LIN {X 0,Y 319.561,Z 300.675,A -85,B 0,C 180,E1 -15416.089,E2 -15416.089} C_VEL
LIN {X 0,Y 319.531,Z 300.681,A -85,B 0,C 180,E1 -15418.933,E2 -15418.933} C_VEL
LIN {X 0,Y 319.51,Z 300.685,A -85,B 0,C 180,E1 -15421.858,E2 -15421.858} C_VEL
LIN {X 0,Y 319.563,Z 300.679,A -85,B 0,C 180,E1 -15425.537,E2 -15425.537} C_VEL
LIN {X 0,Y 319.54,Z 300.681,A -85,B 0,C 180,E1 -15429.663,E2 -15429.663} C_VEL
LIN {X 0,Y 319.497,Z 300.683,A -85,B 0,C 180,E1 -15433.455,E2 -15433.455} C_VEL
LIN {X 0,Y 319.513,Z 300.681,A -85,B 0,C 180,E1 -15437.183,E2 -15437.183} C_VEL
LIN {X 0,Y 319.517,Z 300.684,A -85,B 0,C 180,E1 -15440.366,E2 -15440.366} C_VEL
LIN {X 0,Y 319.508,Z 300.682,A -85,B 0,C 180,E1 -15442.667,E2 -15442.667} C_VEL
LIN {X 0,Y 318.824,Z 300.768,A -85,B 0,C 180,E1 -15443.72,E2 -15443.72} C_VEL
LIN {X 0,Y 315.952,Z 301.126,A -85,B 0,C 180,E1 -15445.434,E2 -15445.434} C_VEL
LIN {X 0,Y 313.541,Z 301.429,A -85,B 0,C 180,E1 -15446.823,E2 -15446.823} C_VEL
LIN {X 0,Y 312.529,Z 301.551,A -85,B 0,C 180,E1 -15447.899,E2 -15447.899} C_VEL
LIN {X 0,Y 312.458,Z 301.56,A -85,B 0,C 180,E1 -15448.263,E2 -15448.263} C_VEL
LIN {X 0,Y 312.537,Z 301.551,A -85,B 0,C 180,E1 -15451.82,E2 -15451.82} C_VEL
LIN {X 0,Y 312.546,Z 301.549,A -85,B 0,C 180,E1 -15454.707,E2 -15454.707} C_VEL
LIN {X 0,Y 312.477,Z 301.558,A -85,B 0,C 180,E1 -15458.908,E2 -15458.908} C_VEL
LIN {X 0,Y 312.519,Z 301.557,A -85,B 0,C 180,E1 -15461.648,E2 -15461.648} C_VEL
LIN {X 0,Y 312.64,Z 301.539,A -85,B 0,C 180,E1 -15465.683,E2 -15465.683} C_VEL
LIN {X 0,Y 312.653,Z 301.536,A -85,B 0,C 180,E1 -15469.64,E2 -15469.64} C_VEL
LIN {X 0,Y 312.798,Z 301.522,A -85,B 0,C 180,E1 -15472.252,E2 -15472.252} C_VEL
LIN {X 0,Y 312.67,Z 301.537,A -85,B 0,C 180,E1 -15474.841,E2 -15474.841} C_VEL
LIN {X 0,Y 312.911,Z 301.504,A -85,B 0,C 180,E1 -15477.425,E2 -15477.425} C_VEL
LIN {X 0,Y 313.034,Z 301.488,A -85,B 0,C 180,E1 -15479.999,E2 -15479.999} C_VEL
LIN {X 0,Y 312.889,Z 301.508,A -85,B 0,C 180,E1 -15482.574,E2 -15482.574} C_VEL
LIN {X 0,Y 312.851,Z 301.511,A -85,B 0,C 180,E1 -15486.448,E2 -15486.448} C_VEL
LIN {X 0,Y 312.712,Z 301.531,A -85,B 0,C 180,E1 -15489.051,E2 -15489.051} C_VEL
LIN {X 0,Y 312.586,Z 301.545,A -85,B 0,C 180,E1 -15492.992,E2 -15492.992} C_VEL
LIN {X 0,Y 312.584,Z 301.549,A -85,B 0,C 180,E1 -15495.652,E2 -15495.652} C_VEL
LIN {X 0,Y 312.565,Z 301.547,A -85,B 0,C 180,E1 -15499.226,E2 -15499.226} C_VEL
LIN {X 0,Y 312.485,Z 301.558,A -85,B 0,C 180,E1 -15502.783,E2 -15502.783} C_VEL
LIN {X 0,Y 312.543,Z 301.551,A -85,B 0,C 180,E1 -15505.931,E2 -15505.931} C_VEL
LIN {X 0,Y 312.467,Z 301.558,A -85,B 0,C 180,E1 -15509.657,E2 -15509.657} C_VEL
LIN {X 0,Y 312.483,Z 301.557,A -85,B 0,C 180,E1 -15513.692,E2 -15513.692} C_VEL
LIN {X 0,Y 312.483,Z 301.56,A -85,B 0,C 180,E1 -15517.39,E2 -15517.39} C_VEL
LIN {X 0,Y 312.457,Z 301.562,A -85,B 0,C 180,E1 -15520.713,E2 -15520.713} C_VEL
LIN {X 0,Y 312.42,Z 301.565,A -85,B 0,C 180,E1 -15524.214,E2 -15524.214} C_VEL
LIN {X 0,Y 312.455,Z 301.564,A -85,B 0,C 180,E1 -15527.924,E2 -15527.924} C_VEL
LIN {X 0,Y 312.452,Z 301.561,A -85,B 0,C 180,E1 -15530.972,E2 -15530.972} C_VEL
LIN {X 0,Y 312.506,Z 301.558,A -85,B 0,C 180,E1 -15534.224,E2 -15534.224} C_VEL
LIN {X 0,Y 312.538,Z 301.702,A -85,B 0,C 180,E1 -15537.345,E2 -15537.345} C_VEL
LIN {X 0,Y 315.451,Z 314.674,A -85,B 0,C 180,E1 -15540.656,E2 -15540.656} C_VEL
LIN {X 0,Y 318.035,Z 327.462,A -85,B 0,C 180,E1 -15543.776,E2 -15543.776} C_VEL
LIN {X 0,Y 316.395,Z 341.128,A -85,B 0,C 180,E1 -15546.784,E2 -15546.784} C_VEL
LIN {X 0,Y 316.002,Z 344.241,A -85,B 0,C 180,E1 -15547.467,E2 -15547.467} C_VEL
LIN {X 0,Y 318.968,Z 375.008,A -85,B 0,C 180,E1 -15548.473,E2 -15548.473} C_VEL
LIN {X 0,Y 317.217,Z 447.196,A -85,B 0,C 180,E1 -15550.426,E2 -15550.426} C_VEL
LIN {X 0,Y 316.799,Z 456.726,A -85,B 0,C 180,E1 -15550.821,E2 -15550.821} C_VEL
LIN {X 0,Y 316.218,Z 466.459,A -85,B 0,C 180,E1 -15551.373,E2 -15551.373} C_VEL
LIN {X 0,Y 315.573,Z 475.191,A -85,B 0,C 180,E1 -15552.005,E2 -15552.005} C_VEL
LIN {X 0,Y 314.745,Z 485.58,A -85,B 0,C 180,E1 -15552.963,E2 -15552.963} C_VEL
LIN {X 0,Y 314.066,Z 494.12,A -85,B 0,C 180,E1 -15553.928,E2 -15553.928} C_VEL
LIN {X 0,Y 313.237,Z 502.921,A -85,B 0,C 180,E1 -15555.13,E2 -15555.13} C_VEL
LIN {X 0,Y 312.614,Z 510.419,A -85,B 0,C 180,E1 -15556.35,E2 -15556.35} C_VEL
LIN {X 0,Y 312.124,Z 517.206,A -85,B 0,C 180,E1 -15557.652,E2 -15557.652} C_VEL
LIN {X 0,Y 311.555,Z 524.228,A -85,B 0,C 180,E1 -15559.278,E2 -15559.278} C_VEL
LIN {X 0,Y 311.202,Z 530.038,A -85,B 0,C 180,E1 -15560.908,E2 -15560.908} C_VEL
LIN {X 0,Y 311.005,Z 535.594,A -85,B 0,C 180,E1 -15562.864,E2 -15562.864} C_VEL
LIN {X 0,Y 310.947,Z 538.236,A -85,B 0,C 180,E1 -15563.973,E2 -15563.973} C_VEL
LIN {X 0,Y 310.901,Z 542.132,A -85,B 0,C 180,E1 -15566.114,E2 -15566.114} C_VEL
LIN {X 0,Y 310.892,Z 543.757,A -85,B 0,C 180,E1 -15567.412,E2 -15567.412} C_VEL
LIN {X 0,Y 311.028,Z 544.971,A -85,B 0,C 180,E1 -15568.708,E2 -15568.708} C_VEL
LIN {X 0,Y 311.069,Z 545.826,A -85,B 0,C 180,E1 -15570.003,E2 -15570.003} C_VEL
LIN {X 0,Y 310.784,Z 545.923,A -85,B 0,C 180,E1 -15572.595,E2 -15572.595} C_VEL
LIN {X 0,Y 310.77,Z 545.451,A -85,B 0,C 180,E1 -15573.892,E2 -15573.892} C_VEL
LIN {X 0,Y 310.772,Z 543.93,A -85,B 0,C 180,E1 -15575.713,E2 -15575.713} C_VEL
LIN {X 0,Y 310.976,Z 541.143,A -85,B 0,C 180,E1 -15577.795,E2 -15577.795} C_VEL
LIN {X 0,Y 311.367,Z 537.429,A -85,B 0,C 180,E1 -15579.748,E2 -15579.748} C_VEL
LIN {X 0,Y 312.047,Z 532.548,A -85,B 0,C 180,E1 -15581.696,E2 -15581.696} C_VEL
LIN {X 0,Y 313.211,Z 526.365,A -85,B 0,C 180,E1 -15583.629,E2 -15583.629} C_VEL
LIN {X 0,Y 314.251,Z 520.119,A -85,B 0,C 180,E1 -15585.236,E2 -15585.236} C_VEL
LIN {X 0,Y 315.608,Z 512.579,A -85,B 0,C 180,E1 -15586.828,E2 -15586.828} C_VEL
LIN {X 0,Y 317.073,Z 504.438,A -85,B 0,C 180,E1 -15588.246,E2 -15588.246} C_VEL
LIN {X 0,Y 318.596,Z 495.771,A -85,B 0,C 180,E1 -15589.491,E2 -15589.491} C_VEL
LIN {X 0,Y 320.051,Z 486.666,A -85,B 0,C 180,E1 -15590.57,E2 -15590.57} C_VEL
LIN {X 0,Y 321.47,Z 477.221,A -85,B 0,C 180,E1 -15591.481,E2 -15591.481} C_VEL
LIN {X 0,Y 322.748,Z 466.457,A -85,B 0,C 180,E1 -15592.316,E2 -15592.316} C_VEL
LIN {X 0,Y 323.729,Z 457.04,A -85,B 0,C 180,E1 -15592.876,E2 -15592.876} C_VEL
LIN {X 0,Y 324.639,Z 446.872,A -85,B 0,C 180,E1 -15593.314,E2 -15593.314} C_VEL
LIN {X 0,Y 325.707,Z 423.932,A -85,B 0,C 180,E1 -15593.992,E2 -15593.992} C_VEL
LIN {X 0,Y 327.83,Z 376.121,A -85,B 0,C 180,E1 -15595.361,E2 -15595.361} C_VEL
LIN {X 0,Y 325.874,Z 360.234,A -85,B 0,C 180,E1 -15596.169,E2 -15596.169} C_VEL
LIN {X 0,Y 322.83,Z 344.326,A -85,B 0,C 180,E1 -15597.151,E2 -15597.151} C_VEL
LIN {X 0,Y 322.58,Z 342.68,A -85,B 0,C 180,E1 -15597.271,E2 -15597.271} C_VEL
LIN {X 0,Y 323.097,Z 338.174,A -85,B 0,C 180,E1 -15598.236,E2 -15598.236} C_VEL
LIN {X 0,Y 321.542,Z 329.706,A -85,B 0,C 180,E1 -15600.485,E2 -15600.485} C_VEL
LIN {X 0,Y 318.939,Z 319.778,A -85,B 0,C 180,E1 -15603.427,E2 -15603.427} C_VEL
LIN {X 0,Y 316.651,Z 312.831,A -85,B 0,C 180,E1 -15605.763,E2 -15605.763} C_VEL
LIN {X 0,Y 313.723,Z 304.747,A -85,B 0,C 180,E1 -15608.846,E2 -15608.846} C_VEL
LIN {X 0,Y 312.479,Z 301.564,A -85,B 0,C 180,E1 -15610.231,E2 -15610.231} C_VEL
LIN {X 0,Y 312.449,Z 301.565,A -85,B 0,C 180,E1 -15613.964,E2 -15613.964} C_VEL
LIN {X 0,Y 312.477,Z 301.559,A -85,B 0,C 180,E1 -15617.918,E2 -15617.918} C_VEL
LIN {X 0,Y 312.53,Z 301.551,A -85,B 0,C 180,E1 -15621.909,E2 -15621.909} C_VEL
LIN {X 0,Y 312.493,Z 301.553,A -85,B 0,C 180,E1 -15625.789,E2 -15625.789} C_VEL
LIN {X 0,Y 312.509,Z 301.548,A -85,B 0,C 180,E1 -15628.853,E2 -15628.853} C_VEL
LIN {X 0,Y 312.559,Z 301.542,A -85,B 0,C 180,E1 -15631.824,E2 -15631.824} C_VEL
LIN {X 0,Y 312.572,Z 301.545,A -85,B 0,C 180,E1 -15634.711,E2 -15634.711} C_VEL
LIN {X 0,Y 312.573,Z 301.551,A -85,B 0,C 180,E1 -15637.529,E2 -15637.529} C_VEL
LIN {X 0,Y 312.621,Z 301.546,A -85,B 0,C 180,E1 -15641.656,E2 -15641.656} C_VEL
LIN {X 0,Y 312.608,Z 301.635,A -85,B 0,C 180,E1 -15644.14,E2 -15644.14} C_VEL
LIN {X 0,Y 315.508,Z 309.164,A -85,B 0,C 180,E1 -15647.13,E2 -15647.13} C_VEL
LIN {X 0,Y 318.415,Z 316.981,A -85,B 0,C 180,E1 -15649.83,E2 -15649.83} C_VEL
LIN {X 0,Y 320.984,Z 325.765,A -85,B 0,C 180,E1 -15652.452,E2 -15652.452} C_VEL
LIN {X 0,Y 322.205,Z 331.817,A -85,B 0,C 180,E1 -15654.054,E2 -15654.054} C_VEL
LIN {X 0,Y 321.513,Z 338.775,A -85,B 0,C 180,E1 -15655.534,E2 -15655.534} C_VEL
LIN {X 0,Y 325.42,Z 357.998,A -85,B 0,C 180,E1 -15656.865,E2 -15656.865} C_VEL
LIN {X 0,Y 327.506,Z 372.724,A -85,B 0,C 180,E1 -15657.73,E2 -15657.73} C_VEL
LIN {X 0,Y 324.419,Z 427.204,A -85,B 0,C 180,E1 -15659.549,E2 -15659.549} C_VEL
LIN {X 0,Y 323.541,Z 438.036,A -85,B 0,C 180,E1 -15660.071,E2 -15660.071} C_VEL
LIN {X 0,Y 322.393,Z 450.107,A -85,B 0,C 180,E1 -15660.906,E2 -15660.906} C_VEL
LIN {X 0,Y 321.132,Z 460.447,A -85,B 0,C 180,E1 -15661.882,E2 -15661.882} C_VEL
LIN {X 0,Y 319.955,Z 468.616,A -85,B 0,C 180,E1 -15662.834,E2 -15662.834} C_VEL
LIN {X 0,Y 318.861,Z 475.526,A -85,B 0,C 180,E1 -15663.792,E2 -15663.792} C_VEL
LIN {X 0,Y 317.505,Z 483.403,A -85,B 0,C 180,E1 -15665.112,E2 -15665.112} C_VEL
LIN {X 0,Y 316.309,Z 489.642,A -85,B 0,C 180,E1 -15666.379,E2 -15666.379} C_VEL
LIN {X 0,Y 315.212,Z 495.003,A -85,B 0,C 180,E1 -15667.689,E2 -15667.689} C_VEL
LIN {X 0,Y 314.311,Z 499.461,A -85,B 0,C 180,E1 -15669.006,E2 -15669.006} C_VEL
LIN {X 0,Y 313.529,Z 503.169,A -85,B 0,C 180,E1 -15670.331,E2 -15670.331} C_VEL
LIN {X 0,Y 312.805,Z 506.225,A -85,B 0,C 180,E1 -15671.667,E2 -15671.667} C_VEL
LIN {X 0,Y 312.252,Z 508.593,A -85,B 0,C 180,E1 -15673.008,E2 -15673.008} C_VEL
LIN {X 0,Y 311.767,Z 510.318,A -85,B 0,C 180,E1 -15674.358,E2 -15674.358} C_VEL
LIN {X 0,Y 311.37,Z 511.487,A -85,B 0,C 180,E1 -15675.716,E2 -15675.716} C_VEL
LIN {X 0,Y 311.102,Z 512.112,A -85,B 0,C 180,E1 -15677.079,E2 -15677.079} C_VEL
LIN {X 0,Y 310.916,Z 512.199,A -85,B 0,C 180,E1 -15678.45,E2 -15678.45} C_VEL
LIN {X 0,Y 310.776,Z 511.681,A -85,B 0,C 180,E1 -15679.83,E2 -15679.83} C_VEL
LIN {X 0,Y 310.787,Z 509.565,A -85,B 0,C 180,E1 -15682.012,E2 -15682.012} C_VEL
LIN {X 0,Y 310.928,Z 507.679,A -85,B 0,C 180,E1 -15683.302,E2 -15683.302} C_VEL
LIN {X 0,Y 311.129,Z 504.922,A -85,B 0,C 180,E1 -15684.702,E2 -15684.702} C_VEL
LIN {X 0,Y 311.489,Z 499.277,A -85,B 0,C 180,E1 -15686.825,E2 -15686.825} C_VEL
LIN {X 0,Y 311.826,Z 494.433,A -85,B 0,C 180,E1 -15688.25,E2 -15688.25} C_VEL
LIN {X 0,Y 312.251,Z 488.495,A -85,B 0,C 180,E1 -15689.681,E2 -15689.681} C_VEL
LIN {X 0,Y 312.852,Z 481.268,A -85,B 0,C 180,E1 -15691.111,E2 -15691.111} C_VEL
LIN {X 0,Y 313.489,Z 473.397,A -85,B 0,C 180,E1 -15692.391,E2 -15692.391} C_VEL
LIN {X 0,Y 314.138,Z 464.159,A -85,B 0,C 180,E1 -15693.623,E2 -15693.623} C_VEL
LIN {X 0,Y 314.847,Z 452.941,A -85,B 0,C 180,E1 -15694.783,E2 -15694.783} C_VEL
LIN {X 0,Y 315.446,Z 444.067,A -85,B 0,C 180,E1 -15695.498,E2 -15695.498} C_VEL
LIN {X 0,Y 315.873,Z 433.915,A -85,B 0,C 180,E1 -15696.13,E2 -15696.13} C_VEL
LIN {X 0,Y 316.224,Z 423.887,A -85,B 0,C 180,E1 -15696.578,E2 -15696.578} C_VEL
LIN {X 0,Y 317.802,Z 367.864,A -85,B 0,C 180,E1 -15698.276,E2 -15698.276} C_VEL
LIN {X 0,Y 314.39,Z 339.94,A -85,B 0,C 180,E1 -15699.315,E2 -15699.315} C_VEL
LIN {X 0,Y 315.823,Z 323.403,A -85,B 0,C 180,E1 -15703.619,E2 -15703.619} C_VEL
LIN {X 0,Y 316.047,Z 319.596,A -85,B 0,C 180,E1 -15704.638,E2 -15704.638} C_VEL
LIN {X 0,Y 313.953,Z 308.571,A -85,B 0,C 180,E1 -15707.814,E2 -15707.814} C_VEL
LIN {X 0,Y 312.499,Z 301.561,A -85,B 0,C 180,E1 -15709.927,E2 -15709.927} C_VEL
LIN {X 0,Y 312.528,Z 301.552,A -85,B 0,C 180,E1 -15714.221,E2 -15714.221} C_VEL
LIN {X 0,Y 312.502,Z 301.556,A -85,B 0,C 180,E1 -15717.334,E2 -15717.334} C_VEL
LIN {X 0,Y 312.486,Z 301.557,A -85,B 0,C 180,E1 -15721.3,E2 -15721.3} C_VEL
LIN {X 0,Y 312.518,Z 301.555,A -85,B 0,C 180,E1 -15724.705,E2 -15724.705} C_VEL
LIN {X 0,Y 312.543,Z 301.549,A -85,B 0,C 180,E1 -15727.525,E2 -15727.525} C_VEL
LIN {X 0,Y 312.571,Z 301.546,A -85,B 0,C 180,E1 -15731.651,E2 -15731.651} C_VEL
LIN {X 0,Y 312.69,Z 301.531,A -85,B 0,C 180,E1 -15735.685,E2 -15735.685} C_VEL
LIN {X 0,Y 312.69,Z 301.533,A -85,B 0,C 180,E1 -15739.64,E2 -15739.64} C_VEL
LIN {X 0,Y 312.801,Z 301.517,A -85,B 0,C 180,E1 -15742.251,E2 -15742.251} C_VEL
LIN {X 0,Y 312.688,Z 301.532,A -85,B 0,C 180,E1 -15744.84,E2 -15744.84} C_VEL
LIN {X 0,Y 312.97,Z 301.496,A -85,B 0,C 180,E1 -15748.711,E2 -15748.711} C_VEL
LIN {X 0,Y 312.969,Z 301.498,A -85,B 0,C 180,E1 -15751.284,E2 -15751.284} C_VEL
LIN {X 0,Y 312.841,Z 301.515,A -85,B 0,C 180,E1 -15756.446,E2 -15756.446} C_VEL
LIN {X 0,Y 312.751,Z 301.524,A -85,B 0,C 180,E1 -15759.047,E2 -15759.047} C_VEL
LIN {X 0,Y 312.633,Z 301.539,A -85,B 0,C 180,E1 -15762.987,E2 -15762.987} C_VEL
LIN {X 0,Y 312.619,Z 301.54,A -85,B 0,C 180,E1 -15765.646,E2 -15765.646} C_VEL
LIN {X 0,Y 312.534,Z 301.551,A -85,B 0,C 180,E1 -15769.708,E2 -15769.708} C_VEL
LIN {X 0,Y 312.515,Z 301.556,A -85,B 0,C 180,E1 -15772.773,E2 -15772.773} C_VEL
LIN {X 0,Y 312.521,Z 301.553,A -85,B 0,C 180,E1 -15775.903,E2 -15775.903} C_VEL
LIN {X 0,Y 312.483,Z 301.56,A -85,B 0,C 180,E1 -15779.65,E2 -15779.65} C_VEL
LIN {X 0,Y 312.505,Z 301.561,A -85,B 0,C 180,E1 -15783.683,E2 -15783.683} C_VEL
LIN {X 0,Y 312.501,Z 301.556,A -85,B 0,C 180,E1 -15787.381,E2 -15787.381} C_VEL
LIN {X 0,Y 312.468,Z 301.559,A -85,B 0,C 180,E1 -15790.704,E2 -15790.704} C_VEL
LIN {X 0,Y 312.427,Z 301.57,A -85,B 0,C 180,E1 -15794.205,E2 -15794.205} C_VEL
LIN {X 0,Y 312.441,Z 301.563,A -85,B 0,C 180,E1 -15797.917,E2 -15797.917} C_VEL
LIN {X 0,Y 312.468,Z 301.562,A -85,B 0,C 180,E1 -15800.966,E2 -15800.966} C_VEL
LIN {X 0,Y 312.498,Z 301.556,A -85,B 0,C 180,E1 -15804.215,E2 -15804.215} C_VEL
LIN {X 0,Y 312.47,Z 301.561,A -85,B 0,C 180,E1 -15807.329,E2 -15807.329} C_VEL
LIN {X 0,Y 312.458,Z 301.56,A -85,B 0,C 180,E1 -15808.263,E2 -15808.263} C_VEL
LIN {X 0,Y 311.806,Z 301.646,A -85,B 0,C 180,E1 -15809.339,E2 -15809.339} C_VEL
LIN {X 0,Y 308.92,Z 302.008,A -85,B 0,C 180,E1 -15811.089,E2 -15811.089} C_VEL
LIN {X 0,Y 306.512,Z 302.307,A -85,B 0,C 180,E1 -15812.509,E2 -15812.509} C_VEL
LIN {X 0,Y 305.551,Z 302.424,A -85,B 0,C 180,E1 -15813.609,E2 -15813.609} C_VEL
LIN {X 0,Y 305.513,Z 302.426,A -85,B 0,C 180,E1 -15813.981,E2 -15813.981} C_VEL
LIN {X 0,Y 305.454,Z 302.433,A -85,B 0,C 180,E1 -15816.974,E2 -15816.974} C_VEL
LIN {X 0,Y 305.472,Z 302.431,A -85,B 0,C 180,E1 -15821.209,E2 -15821.209} C_VEL
LIN {X 0,Y 305.582,Z 302.416,A -85,B 0,C 180,E1 -15825.345,E2 -15825.345} C_VEL
LIN {X 0,Y 305.59,Z 302.416,A -85,B 0,C 180,E1 -15829.397,E2 -15829.397} C_VEL
LIN {X 0,Y 305.741,Z 302.399,A -85,B 0,C 180,E1 -15832.072,E2 -15832.072} C_VEL
LIN {X 0,Y 305.641,Z 302.414,A -85,B 0,C 180,E1 -15834.722,E2 -15834.722} C_VEL
LIN {X 0,Y 305.912,Z 302.38,A -85,B 0,C 180,E1 -15838.683,E2 -15838.683} C_VEL
LIN {X 0,Y 305.909,Z 302.378,A -85,B 0,C 180,E1 -15841.316,E2 -15841.316} C_VEL
LIN {X 0,Y 305.639,Z 302.415,A -85,B 0,C 180,E1 -15845.277,E2 -15845.277} C_VEL
LIN {X 0,Y 305.74,Z 302.398,A -85,B 0,C 180,E1 -15847.927,E2 -15847.927} C_VEL
LIN {X 0,Y 305.555,Z 302.422,A -85,B 0,C 180,E1 -15851.946,E2 -15851.946} C_VEL
LIN {X 0,Y 305.576,Z 302.418,A -85,B 0,C 180,E1 -15855.023,E2 -15855.023} C_VEL
LIN {X 0,Y 305.534,Z 302.422,A -85,B 0,C 180,E1 -15858.785,E2 -15858.785} C_VEL
LIN {X 0,Y 305.446,Z 302.434,A -85,B 0,C 180,E1 -15863.042,E2 -15863.042} C_VEL
LIN {X 0,Y 305.475,Z 302.434,A -85,B 0,C 180,E1 -15866.217,E2 -15866.217} C_VEL
LIN {X 0,Y 305.43,Z 302.436,A -85,B 0,C 180,E1 -15869.043,E2 -15869.043} C_VEL
LIN {X 0,Y 305.398,Z 302.44,A -85,B 0,C 180,E1 -15871.957,E2 -15871.957} C_VEL
LIN {X 0,Y 305.425,Z 302.44,A -85,B 0,C 180,E1 -15875.117,E2 -15875.117} C_VEL
LIN {X 0,Y 305.405,Z 302.44,A -85,B 0,C 180,E1 -15878.53,E2 -15878.53} C_VEL
LIN {X 0,Y 305.396,Z 302.441,A -85,B 0,C 180,E1 -15881.863,E2 -15881.863} C_VEL
LIN {X 0,Y 305.37,Z 302.449,A -85,B 0,C 180,E1 -15885.516,E2 -15885.516} C_VEL
LIN {X 0,Y 305.412,Z 302.44,A -85,B 0,C 180,E1 -15888.147,E2 -15888.147} C_VEL
LIN {X 0,Y 305.43,Z 302.44,A -85,B 0,C 180,E1 -15891.599,E2 -15891.599} C_VEL
LIN {X 0,Y 305.438,Z 302.435,A -85,B 0,C 180,E1 -15894.891,E2 -15894.891} C_VEL
LIN {X 0,Y 305.523,Z 302.623,A -85,B 0,C 180,E1 -15896.99,E2 -15896.99} C_VEL
LIN {X 0,Y 308.337,Z 315.249,A -85,B 0,C 180,E1 -15900.302,E2 -15900.302} C_VEL
LIN {X 0,Y 310.962,Z 328.017,A -85,B 0,C 180,E1 -15903.495,E2 -15903.495} C_VEL
LIN {X 0,Y 310.856,Z 331.099,A -85,B 0,C 180,E1 -15904.207,E2 -15904.207} C_VEL
LIN {X 0,Y 309.07,Z 344.407,A -85,B 0,C 180,E1 -15907.154,E2 -15907.154} C_VEL
LIN {X 0,Y 312.05,Z 375.781,A -85,B 0,C 180,E1 -15908.203,E2 -15908.203} C_VEL
LIN {X 0,Y 310.244,Z 447.06,A -85,B 0,C 180,E1 -15910.183,E2 -15910.183} C_VEL
LIN {X 0,Y 309.818,Z 456.53,A -85,B 0,C 180,E1 -15910.586,E2 -15910.586} C_VEL
LIN {X 0,Y 309.27,Z 465.646,A -85,B 0,C 180,E1 -15911.11,E2 -15911.11} C_VEL
LIN {X 0,Y 308.613,Z 474.48,A -85,B 0,C 180,E1 -15911.757,E2 -15911.757} C_VEL
LIN {X 0,Y 307.777,Z 484.932,A -85,B 0,C 180,E1 -15912.736,E2 -15912.736} C_VEL
LIN {X 0,Y 307.071,Z 493.521,A -85,B 0,C 180,E1 -15913.722,E2 -15913.722} C_VEL
LIN {X 0,Y 306.25,Z 501.887,A -85,B 0,C 180,E1 -15914.876,E2 -15914.876} C_VEL
LIN {X 0,Y 305.678,Z 509.021,A -85,B 0,C 180,E1 -15916.034,E2 -15916.034} C_VEL
LIN {X 0,Y 304.994,Z 517.424,A -85,B 0,C 180,E1 -15917.697,E2 -15917.697} C_VEL
LIN {X 0,Y 304.463,Z 524.347,A -85,B 0,C 180,E1 -15919.362,E2 -15919.362} C_VEL
LIN {X 0,Y 304.155,Z 529.073,A -85,B 0,C 180,E1 -15920.695,E2 -15920.695} C_VEL
LIN {X 0,Y 303.931,Z 534.749,A -85,B 0,C 180,E1 -15922.697,E2 -15922.697} C_VEL
LIN {X 0,Y 303.855,Z 539.118,A -85,B 0,C 180,E1 -15924.695,E2 -15924.695} C_VEL
LIN {X 0,Y 303.839,Z 541.438,A -85,B 0,C 180,E1 -15926.024,E2 -15926.024} C_VEL
LIN {X 0,Y 303.937,Z 544.415,A -85,B 0,C 180,E1 -15928.678,E2 -15928.678} C_VEL
LIN {X 0,Y 303.992,Z 545.32,A -85,B 0,C 180,E1 -15930.003,E2 -15930.003} C_VEL
LIN {X 0,Y 303.702,Z 545.548,A -85,B 0,C 180,E1 -15932.655,E2 -15932.655} C_VEL
LIN {X 0,Y 303.679,Z 545.104,A -85,B 0,C 180,E1 -15933.983,E2 -15933.983} C_VEL
LIN {X 0,Y 303.724,Z 542.731,A -85,B 0,C 180,E1 -15936.646,E2 -15936.646} C_VEL
LIN {X 0,Y 304.028,Z 539.813,A -85,B 0,C 180,E1 -15938.644,E2 -15938.644} C_VEL
LIN {X 0,Y 304.566,Z 535.836,A -85,B 0,C 180,E1 -15940.64,E2 -15940.64} C_VEL
LIN {X 0,Y 305.07,Z 532.626,A -85,B 0,C 180,E1 -15941.968,E2 -15941.968} C_VEL
LIN {X 0,Y 306.304,Z 526.595,A -85,B 0,C 180,E1 -15943.942,E2 -15943.942} C_VEL
LIN {X 0,Y 307.625,Z 519.026,A -85,B 0,C 180,E1 -15945.913,E2 -15945.913} C_VEL
LIN {X 0,Y 308.846,Z 513.058,A -85,B 0,C 180,E1 -15947.208,E2 -15947.208} C_VEL
LIN {X 0,Y 310.591,Z 504.071,A -85,B 0,C 180,E1 -15948.812,E2 -15948.812} C_VEL
LIN {X 0,Y 312.168,Z 495.483,A -85,B 0,C 180,E1 -15950.081,E2 -15950.081} C_VEL
LIN {X 0,Y 313.743,Z 486.47,A -85,B 0,C 180,E1 -15951.175,E2 -15951.175} C_VEL
LIN {X 0,Y 315.206,Z 477.12,A -85,B 0,C 180,E1 -15952.102,E2 -15952.102} C_VEL
LIN {X 0,Y 316.567,Z 466.412,A -85,B 0,C 180,E1 -15952.949,E2 -15952.949} C_VEL
LIN {X 0,Y 317.715,Z 456.324,A -85,B 0,C 180,E1 -15953.55,E2 -15953.55} C_VEL
LIN {X 0,Y 318.616,Z 446.046,A -85,B 0,C 180,E1 -15953.997,E2 -15953.997} C_VEL
LIN {X 0,Y 322.008,Z 377.404,A -85,B 0,C 180,E1 -15956.037,E2 -15956.037} C_VEL
LIN {X 0,Y 320.17,Z 361.869,A -85,B 0,C 180,E1 -15956.854,E2 -15956.854} C_VEL
LIN {X 0,Y 317.028,Z 345.072,A -85,B 0,C 180,E1 -15957.945,E2 -15957.945} C_VEL
LIN {X 0,Y 316.537,Z 342.717,A -85,B 0,C 180,E1 -15958.115,E2 -15958.115} C_VEL
LIN {X 0,Y 316.731,Z 341.02,A -85,B 0,C 180,E1 -15958.493,E2 -15958.493} C_VEL
LIN {X 0,Y 315.465,Z 333.668,A -85,B 0,C 180,E1 -15960.474,E2 -15960.474} C_VEL
LIN {X 0,Y 313.265,Z 324.624,A -85,B 0,C 180,E1 -15963.2,E2 -15963.2} C_VEL
LIN {X 0,Y 311.101,Z 317.62,A -85,B 0,C 180,E1 -15965.585,E2 -15965.585} C_VEL
LIN {X 0,Y 308.345,Z 309.992,A -85,B 0,C 180,E1 -15968.555,E2 -15968.555} C_VEL
LIN {X 0,Y 306.323,Z 305.083,A -85,B 0,C 180,E1 -15970.79,E2 -15970.79} C_VEL
LIN {X 0,Y 305.445,Z 302.44,A -85,B 0,C 180,E1 -15972.128,E2 -15972.128} C_VEL
LIN {X 0,Y 305.416,Z 302.441,A -85,B 0,C 180,E1 -15976.344,E2 -15976.344} C_VEL
LIN {X 0,Y 305.451,Z 302.433,A -85,B 0,C 180,E1 -15979.892,E2 -15979.892} C_VEL
LIN {X 0,Y 305.487,Z 302.43,A -85,B 0,C 180,E1 -15983.627,E2 -15983.627} C_VEL
LIN {X 0,Y 305.452,Z 302.427,A -85,B 0,C 180,E1 -15986.482,E2 -15986.482} C_VEL
LIN {X 0,Y 305.448,Z 302.425,A -85,B 0,C 180,E1 -15989.59,E2 -15989.59} C_VEL
LIN {X 0,Y 305.502,Z 302.424,A -85,B 0,C 180,E1 -15992.608,E2 -15992.608} C_VEL
LIN {X 0,Y 305.496,Z 302.431,A -85,B 0,C 180,E1 -15995.539,E2 -15995.539} C_VEL
LIN {X 0,Y 305.517,Z 302.43,A -85,B 0,C 180,E1 -15999.816,E2 -15999.816} C_VEL
LIN {X 0,Y 305.569,Z 302.583,A -85,B 0,C 180,E1 -16002.344,E2 -16002.344} C_VEL
LIN {X 0,Y 308.406,Z 309.447,A -85,B 0,C 180,E1 -16005.484,E2 -16005.484} C_VEL
LIN {X 0,Y 311.376,Z 317.454,A -85,B 0,C 180,E1 -16008.519,E2 -16008.519} C_VEL
LIN {X 0,Y 313.789,Z 324.958,A -85,B 0,C 180,E1 -16010.981,E2 -16010.981} C_VEL
LIN {X 0,Y 315.403,Z 331.797,A -85,B 0,C 180,E1 -16012.961,E2 -16012.961} C_VEL
LIN {X 0,Y 315.962,Z 335.523,A -85,B 0,C 180,E1 -16013.936,E2 -16013.936} C_VEL
LIN {X 0,Y 315.517,Z 338.867,A -85,B 0,C 180,E1 -16014.649,E2 -16014.649} C_VEL
LIN {X 0,Y 319.253,Z 357.274,A -85,B 0,C 180,E1 -16016.016,E2 -16016.016} C_VEL
LIN {X 0,Y 321.567,Z 372.824,A -85,B 0,C 180,E1 -16016.984,E2 -16016.984} C_VEL
LIN {X 0,Y 318.307,Z 428.295,A -85,B 0,C 180,E1 -16018.924,E2 -16018.924} C_VEL
LIN {X 0,Y 317.36,Z 439.474,A -85,B 0,C 180,E1 -16019.488,E2 -16019.488} C_VEL
LIN {X 0,Y 316.092,Z 451.515,A -85,B 0,C 180,E1 -16020.369,E2 -16020.369} C_VEL
LIN {X 0,Y 314.881,Z 460.932,A -85,B 0,C 180,E1 -16021.28,E2 -16021.28} C_VEL
LIN {X 0,Y 313.636,Z 469.098,A -85,B 0,C 180,E1 -16022.248,E2 -16022.248} C_VEL
LIN {X 0,Y 312.274,Z 477.012,A -85,B 0,C 180,E1 -16023.388,E2 -16023.388} C_VEL
LIN {X 0,Y 310.933,Z 484.094,A -85,B 0,C 180,E1 -16024.621,E2 -16024.621} C_VEL
LIN {X 0,Y 309.723,Z 490.025,A -85,B 0,C 180,E1 -16025.861,E2 -16025.861} C_VEL
LIN {X 0,Y 308.55,Z 495.39,A -85,B 0,C 180,E1 -16027.197,E2 -16027.197} C_VEL
LIN {X 0,Y 307.568,Z 499.866,A -85,B 0,C 180,E1 -16028.542,E2 -16028.542} C_VEL
LIN {X 0,Y 306.334,Z 505.157,A -85,B 0,C 180,E1 -16030.577,E2 -16030.577} C_VEL
LIN {X 0,Y 305.342,Z 509.017,A -85,B 0,C 180,E1 -16032.631,E2 -16032.631} C_VEL
LIN {X 0,Y 304.588,Z 511.445,A -85,B 0,C 180,E1 -16034.704,E2 -16034.704} C_VEL
LIN {X 0,Y 304.217,Z 512.362,A -85,B 0,C 180,E1 -16036.095,E2 -16036.095} C_VEL
LIN {X 0,Y 303.817,Z 512.54,A -85,B 0,C 180,E1 -16038.49,E2 -16038.49} C_VEL
LIN {X 0,Y 303.673,Z 511.58,A -85,B 0,C 180,E1 -16040.314,E2 -16040.314} C_VEL
LIN {X 0,Y 303.711,Z 509.475,A -85,B 0,C 180,E1 -16042.245,E2 -16042.245} C_VEL
LIN {X 0,Y 303.911,Z 506.803,A -85,B 0,C 180,E1 -16043.873,E2 -16043.873} C_VEL
LIN {X 0,Y 304.158,Z 502.737,A -85,B 0,C 180,E1 -16045.696,E2 -16045.696} C_VEL
LIN {X 0,Y 304.522,Z 497.521,A -85,B 0,C 180,E1 -16047.49,E2 -16047.49} C_VEL
LIN {X 0,Y 305.073,Z 490.766,A -85,B 0,C 180,E1 -16049.311,E2 -16049.311} C_VEL
LIN {X 0,Y 305.59,Z 483.904,A -85,B 0,C 180,E1 -16050.779,E2 -16050.779} C_VEL
LIN {X 0,Y 306.277,Z 475.477,A -85,B 0,C 180,E1 -16052.244,E2 -16052.244} C_VEL
LIN {X 0,Y 306.862,Z 467.81,A -85,B 0,C 180,E1 -16053.345,E2 -16053.345} C_VEL
LIN {X 0,Y 307.414,Z 460.172,A -85,B 0,C 180,E1 -16054.262,E2 -16054.262} C_VEL
LIN {X 0,Y 307.989,Z 450.804,A -85,B 0,C 180,E1 -16055.183,E2 -16055.183} C_VEL
LIN {X 0,Y 308.572,Z 441.451,A -85,B 0,C 180,E1 -16055.908,E2 -16055.908} C_VEL
LIN {X 0,Y 309.096,Z 429.632,A -85,B 0,C 180,E1 -16056.595,E2 -16056.595} C_VEL
LIN {X 0,Y 309.611,Z 412.785,A -85,B 0,C 180,E1 -16057.185,E2 -16057.185} C_VEL
LIN {X 0,Y 310.82,Z 367.928,A -85,B 0,C 180,E1 -16058.565,E2 -16058.565} C_VEL
LIN {X 0,Y 307.434,Z 339.917,A -85,B 0,C 180,E1 -16059.644,E2 -16059.644} C_VEL
LIN {X 0,Y 308.924,Z 323.687,A -85,B 0,C 180,E1 -16063.958,E2 -16063.958} C_VEL
LIN {X 0,Y 308.854,Z 319.433,A -85,B 0,C 180,E1 -16065.14,E2 -16065.14} C_VEL
LIN {X 0,Y 306.715,Z 308.538,A -85,B 0,C 180,E1 -16068.358,E2 -16068.358} C_VEL
LIN {X 0,Y 305.467,Z 302.435,A -85,B 0,C 180,E1 -16070.271,E2 -16070.271} C_VEL
LIN {X 0,Y 305.46,Z 302.437,A -85,B 0,C 180,E1 -16073.638,E2 -16073.638} C_VEL
LIN {X 0,Y 305.465,Z 302.432,A -85,B 0,C 180,E1 -16076.484,E2 -16076.484} C_VEL
LIN {X 0,Y 305.418,Z 302.439,A -85,B 0,C 180,E1 -16079.586,E2 -16079.586} C_VEL
LIN {X 0,Y 305.443,Z 302.436,A -85,B 0,C 180,E1 -16082.601,E2 -16082.601} C_VEL
LIN {X 0,Y 305.442,Z 302.434,A -85,B 0,C 180,E1 -16085.533,E2 -16085.533} C_VEL
LIN {X 0,Y 305.485,Z 302.429,A -85,B 0,C 180,E1 -16089.812,E2 -16089.812} C_VEL
LIN {X 0,Y 305.556,Z 302.42,A -85,B 0,C 180,E1 -16093.977,E2 -16093.977} C_VEL
LIN {X 0,Y 305.591,Z 302.418,A -85,B 0,C 180,E1 -16096.703,E2 -16096.703} C_VEL
LIN {X 0,Y 305.758,Z 302.401,A -85,B 0,C 180,E1 -16101.26,E2 -16101.26} C_VEL
LIN {X 0,Y 305.789,Z 302.396,A -85,B 0,C 180,E1 -16103.399,E2 -16103.399} C_VEL
LIN {X 0,Y 305.938,Z 302.372,A -85,B 0,C 180,E1 -16108.681,E2 -16108.681} C_VEL
LIN {X 0,Y 305.937,Z 302.374,A -85,B 0,C 180,E1 -16111.314,E2 -16111.314} C_VEL
LIN {X 0,Y 305.786,Z 302.393,A -85,B 0,C 180,E1 -16116.595,E2 -16116.595} C_VEL
LIN {X 0,Y 305.695,Z 302.402,A -85,B 0,C 180,E1 -16119.257,E2 -16119.257} C_VEL
LIN {X 0,Y 305.585,Z 302.416,A -85,B 0,C 180,E1 -16123.292,E2 -16123.292} C_VEL
LIN {X 0,Y 305.548,Z 302.422,A -85,B 0,C 180,E1 -16126.018,E2 -16126.018} C_VEL
LIN {X 0,Y 305.479,Z 302.43,A -85,B 0,C 180,E1 -16130.183,E2 -16130.183} C_VEL
LIN {X 0,Y 305.466,Z 302.432,A -85,B 0,C 180,E1 -16134.459,E2 -16134.459} C_VEL
LIN {X 0,Y 305.446,Z 302.439,A -85,B 0,C 180,E1 -16137.393,E2 -16137.393} C_VEL
LIN {X 0,Y 305.417,Z 302.436,A -85,B 0,C 180,E1 -16140.408,E2 -16140.408} C_VEL
LIN {X 0,Y 305.449,Z 302.436,A -85,B 0,C 180,E1 -16144.073,E2 -16144.073} C_VEL
LIN {X 0,Y 305.439,Z 302.434,A -85,B 0,C 180,E1 -16146.737,E2 -16146.737} C_VEL
LIN {X 0,Y 305.434,Z 302.436,A -85,B 0,C 180,E1 -16150.594,E2 -16150.594} C_VEL
LIN {X 0,Y 305.402,Z 302.44,A -85,B 0,C 180,E1 -16153.65,E2 -16153.65} C_VEL
LIN {X 0,Y 305.416,Z 302.437,A -85,B 0,C 180,E1 -16157.412,E2 -16157.412} C_VEL
LIN {X 0,Y 305.431,Z 302.436,A -85,B 0,C 180,E1 -16159.887,E2 -16159.887} C_VEL
LIN {X 0,Y 305.432,Z 302.435,A -85,B 0,C 180,E1 -16163.632,E2 -16163.632} C_VEL
LIN {X 0,Y 305.432,Z 302.437,A -85,B 0,C 180,E1 -16166.478,E2 -16166.478} C_VEL
LIN {X 0,Y 305.46,Z 302.435,A -85,B 0,C 180,E1 -16170.947,E2 -16170.947} C_VEL
LIN {X 0,Y 305.513,Z 302.426,A -85,B 0,C 180,E1 -16173.981,E2 -16173.981} C_VEL
LIN {X 0,Y 305.27,Z 302.458,A -85,B 0,C 180,E1 -16174.716,E2 -16174.716} C_VEL
LIN {X 0,Y 303.949,Z 302.625,A -85,B 0,C 180,E1 -16175.802,E2 -16175.802} C_VEL
LIN {X 0,Y 299.522,Z 303.172,A -85,B 0,C 180,E1 -16178.321,E2 -16178.321} C_VEL
LIN {X 0,Y 298.453,Z 303.308,A -85,B 0,C 180,E1 -16179.447,E2 -16179.447} C_VEL
LIN {X 0,Y 298.376,Z 303.314,A -85,B 0,C 180,E1 -16179.829,E2 -16179.829} C_VEL
LIN {X 0,Y 298.437,Z 303.309,A -85,B 0,C 180,E1 -16183.584,E2 -16183.584} C_VEL
LIN {X 0,Y 298.5,Z 303.302,A -85,B 0,C 180,E1 -16186.381,E2 -16186.381} C_VEL
LIN {X 0,Y 298.679,Z 303.277,A -85,B 0,C 180,E1 -16191.161,E2 -16191.161} C_VEL
LIN {X 0,Y 298.738,Z 303.269,A -85,B 0,C 180,E1 -16193.244,E2 -16193.244} C_VEL
LIN {X 0,Y 298.806,Z 303.262,A -85,B 0,C 180,E1 -16197.303,E2 -16197.303} C_VEL
LIN {X 0,Y 298.946,Z 303.243,A -85,B 0,C 180,E1 -16199.999,E2 -16199.999} C_VEL
LIN {X 0,Y 298.789,Z 303.265,A -85,B 0,C 180,E1 -16202.696,E2 -16202.696} C_VEL
LIN {X 0,Y 298.736,Z 303.271,A -85,B 0,C 180,E1 -16206.755,E2 -16206.755} C_VEL
LIN {X 0,Y 298.586,Z 303.293,A -85,B 0,C 180,E1 -16209.483,E2 -16209.483} C_VEL
LIN {X 0,Y 298.502,Z 303.304,A -85,B 0,C 180,E1 -16213.617,E2 -16213.617} C_VEL
LIN {X 0,Y 298.484,Z 303.302,A -85,B 0,C 180,E1 -16216.412,E2 -16216.412} C_VEL
LIN {X 0,Y 298.455,Z 303.307,A -85,B 0,C 180,E1 -16219.648,E2 -16219.648} C_VEL
LIN {X 0,Y 298.387,Z 303.313,A -85,B 0,C 180,E1 -16223.603,E2 -16223.603} C_VEL
LIN {X 0,Y 298.419,Z 303.313,A -85,B 0,C 180,E1 -16226.58,E2 -16226.58} C_VEL
LIN {X 0,Y 298.364,Z 303.315,A -85,B 0,C 180,E1 -16229.646,E2 -16229.646} C_VEL
LIN {X 0,Y 298.355,Z 303.323,A -85,B 0,C 180,E1 -16232.804,E2 -16232.804} C_VEL
LIN {X 0,Y 298.408,Z 303.314,A -85,B 0,C 180,E1 -16236.81,E2 -16236.81} C_VEL
LIN {X 0,Y 298.35,Z 303.322,A -85,B 0,C 180,E1 -16241.09,E2 -16241.09} C_VEL
LIN {X 0,Y 298.37,Z 303.319,A -85,B 0,C 180,E1 -16243.107,E2 -16243.107} C_VEL
LIN {X 0,Y 298.377,Z 303.315,A -85,B 0,C 180,E1 -16246.925,E2 -16246.925} C_VEL
LIN {X 0,Y 298.365,Z 303.316,A -85,B 0,C 180,E1 -16251.014,E2 -16251.014} C_VEL
LIN {X 0,Y 298.381,Z 303.319,A -85,B 0,C 180,E1 -16253.933,E2 -16253.933} C_VEL
LIN {X 0,Y 298.453,Z 303.444,A -85,B 0,C 180,E1 -16256.61,E2 -16256.61} C_VEL
LIN {X 0,Y 301.463,Z 316.996,A -85,B 0,C 180,E1 -16260.24,E2 -16260.24} C_VEL
LIN {X 0,Y 303.853,Z 328.541,A -85,B 0,C 180,E1 -16263.196,E2 -16263.196} C_VEL
LIN {X 0,Y 303.919,Z 331.646,A -85,B 0,C 180,E1 -16263.942,E2 -16263.942} C_VEL
LIN {X 0,Y 302.16,Z 344.254,A -85,B 0,C 180,E1 -16266.822,E2 -16266.822} C_VEL
LIN {X 0,Y 305.138,Z 376.347,A -85,B 0,C 180,E1 -16267.922,E2 -16267.922} C_VEL
LIN {X 0,Y 303.297,Z 446.293,A -85,B 0,C 180,E1 -16269.931,E2 -16269.931} C_VEL
LIN {X 0,Y 302.863,Z 455.875,A -85,B 0,C 180,E1 -16270.343,E2 -16270.343} C_VEL
LIN {X 0,Y 302.257,Z 465.637,A -85,B 0,C 180,E1 -16270.919,E2 -16270.919} C_VEL
LIN {X 0,Y 301.5,Z 475.312,A -85,B 0,C 180,E1 -16271.663,E2 -16271.663} C_VEL
LIN {X 0,Y 300.689,Z 485.557,A -85,B 0,C 180,E1 -16272.667,E2 -16272.667} C_VEL
LIN {X 0,Y 299.981,Z 493.981,A -85,B 0,C 180,E1 -16273.676,E2 -16273.676} C_VEL
LIN {X 0,Y 299.173,Z 501.968,A -85,B 0,C 180,E1 -16274.816,E2 -16274.816} C_VEL
LIN {X 0,Y 298.559,Z 509.24,A -85,B 0,C 180,E1 -16276.042,E2 -16276.042} C_VEL
LIN {X 0,Y 297.864,Z 517.544,A -85,B 0,C 180,E1 -16277.744,E2 -16277.744} C_VEL
LIN {X 0,Y 297.359,Z 524.388,A -85,B 0,C 180,E1 -16279.449,E2 -16279.449} C_VEL
LIN {X 0,Y 297.012,Z 530.025,A -85,B 0,C 180,E1 -16281.156,E2 -16281.156} C_VEL
LIN {X 0,Y 296.871,Z 533.861,A -85,B 0,C 180,E1 -16282.522,E2 -16282.522} C_VEL
LIN {X 0,Y 296.788,Z 538.353,A -85,B 0,C 180,E1 -16284.568,E2 -16284.568} C_VEL
LIN {X 0,Y 296.779,Z 540.685,A -85,B 0,C 180,E1 -16285.929,E2 -16285.929} C_VEL
LIN {X 0,Y 296.846,Z 543.856,A -85,B 0,C 180,E1 -16288.646,E2 -16288.646} C_VEL
LIN {X 0,Y 296.937,Z 544.775,A -85,B 0,C 180,E1 -16290.003,E2 -16290.003} C_VEL
LIN {X 0,Y 296.622,Z 545.172,A -85,B 0,C 180,E1 -16292.719,E2 -16292.719} C_VEL
LIN {X 0,Y 296.592,Z 544.728,A -85,B 0,C 180,E1 -16294.079,E2 -16294.079} C_VEL
LIN {X 0,Y 296.648,Z 542.54,A -85,B 0,C 180,E1 -16296.805,E2 -16296.805} C_VEL
LIN {X 0,Y 296.984,Z 539.734,A -85,B 0,C 180,E1 -16298.85,E2 -16298.85} C_VEL
LIN {X 0,Y 297.571,Z 535.855,A -85,B 0,C 180,E1 -16300.893,E2 -16300.893} C_VEL
LIN {X 0,Y 298.514,Z 530.802,A -85,B 0,C 180,E1 -16302.926,E2 -16302.926} C_VEL
LIN {X 0,Y 299.607,Z 525.62,A -85,B 0,C 180,E1 -16304.607,E2 -16304.607} C_VEL
LIN {X 0,Y 300.975,Z 518.413,A -85,B 0,C 180,E1 -16306.518,E2 -16306.518} C_VEL
LIN {X 0,Y 302.411,Z 511.941,A -85,B 0,C 180,E1 -16307.935,E2 -16307.935} C_VEL
LIN {X 0,Y 304.132,Z 503.871,A -85,B 0,C 180,E1 -16309.402,E2 -16309.402} C_VEL
LIN {X 0,Y 305.791,Z 495.308,A -85,B 0,C 180,E1 -16310.694,E2 -16310.694} C_VEL
LIN {X 0,Y 307.461,Z 486.322,A -85,B 0,C 180,E1 -16311.805,E2 -16311.805} C_VEL
LIN {X 0,Y 309.001,Z 477.013,A -85,B 0,C 180,E1 -16312.747,E2 -16312.747} C_VEL
LIN {X 0,Y 310.428,Z 466.441,A -85,B 0,C 180,E1 -16313.606,E2 -16313.606} C_VEL
LIN {X 0,Y 311.726,Z 455.858,A -85,B 0,C 180,E1 -16314.252,E2 -16314.252} C_VEL
LIN {X 0,Y 312.682,Z 445.697,A -85,B 0,C 180,E1 -16314.704,E2 -16314.704} C_VEL
LIN {X 0,Y 315.413,Z 394.829,A -85,B 0,C 180,E1 -16316.248,E2 -16316.248} C_VEL
LIN {X 0,Y 316.141,Z 377.744,A -85,B 0,C 180,E1 -16316.795,E2 -16316.795} C_VEL
LIN {X 0,Y 314.441,Z 362.812,A -85,B 0,C 180,E1 -16317.619,E2 -16317.619} C_VEL
LIN {X 0,Y 311.231,Z 345.592,A -85,B 0,C 180,E1 -16318.805,E2 -16318.805} C_VEL
LIN {X 0,Y 310.276,Z 342.536,A -85,B 0,C 180,E1 -16319.104,E2 -16319.104} C_VEL
LIN {X 0,Y 308.622,Z 333.962,A -85,B 0,C 180,E1 -16321.584,E2 -16321.584} C_VEL
LIN {X 0,Y 306.451,Z 325.416,A -85,B 0,C 180,E1 -16324.351,E2 -16324.351} C_VEL
LIN {X 0,Y 303.652,Z 316.826,A -85,B 0,C 180,E1 -16327.573,E2 -16327.573} C_VEL
LIN {X 0,Y 301.311,Z 310.626,A -85,B 0,C 180,E1 -16330.322,E2 -16330.322} C_VEL
LIN {X 0,Y 299.694,Z 306.607,A -85,B 0,C 180,E1 -16332.382,E2 -16332.382} C_VEL
LIN {X 0,Y 298.366,Z 303.321,A -85,B 0,C 180,E1 -16334.319,E2 -16334.319} C_VEL
LIN {X 0,Y 298.395,Z 303.317,A -85,B 0,C 180,E1 -16336.92,E2 -16336.92} C_VEL
LIN {X 0,Y 298.414,Z 303.312,A -85,B 0,C 180,E1 -16341.001,E2 -16341.001} C_VEL
LIN {X 0,Y 298.419,Z 303.308,A -85,B 0,C 180,E1 -16343.931,E2 -16343.931} C_VEL
LIN {X 0,Y 298.382,Z 303.308,A -85,B 0,C 180,E1 -16347.984,E2 -16347.984} C_VEL
LIN {X 0,Y 298.447,Z 303.299,A -85,B 0,C 180,E1 -16351.903,E2 -16351.903} C_VEL
LIN {X 0,Y 298.47,Z 303.303,A -85,B 0,C 180,E1 -16354.923,E2 -16354.923} C_VEL
LIN {X 0,Y 298.444,Z 303.309,A -85,B 0,C 180,E1 -16359.316,E2 -16359.316} C_VEL
LIN {X 0,Y 298.516,Z 303.432,A -85,B 0,C 180,E1 -16360.119,E2 -16360.119} C_VEL
LIN {X 0,Y 300.656,Z 308.802,A -85,B 0,C 180,E1 -16363.012,E2 -16363.012} C_VEL
LIN {X 0,Y 302.692,Z 313.449,A -85,B 0,C 180,E1 -16365.203,E2 -16365.203} C_VEL
LIN {X 0,Y 305.924,Z 322.541,A -85,B 0,C 180,E1 -16368.74,E2 -16368.74} C_VEL
LIN {X 0,Y 308.314,Z 330.481,A -85,B 0,C 180,E1 -16371.364,E2 -16371.364} C_VEL
LIN {X 0,Y 309.705,Z 337.936,A -85,B 0,C 180,E1 -16373.486,E2 -16373.486} C_VEL
LIN {X 0,Y 309.607,Z 338.993,A -85,B 0,C 180,E1 -16373.729,E2 -16373.729} C_VEL
LIN {X 0,Y 313.558,Z 358.621,A -85,B 0,C 180,E1 -16375.255,E2 -16375.255} C_VEL
LIN {X 0,Y 315.792,Z 374.119,A -85,B 0,C 180,E1 -16376.274,E2 -16376.274} C_VEL
LIN {X 0,Y 312.364,Z 428.907,A -85,B 0,C 180,E1 -16378.228,E2 -16378.228} C_VEL
LIN {X 0,Y 311.287,Z 440.812,A -85,B 0,C 180,E1 -16378.856,E2 -16378.856} C_VEL
LIN {X 0,Y 309.918,Z 452.405,A -85,B 0,C 180,E1 -16379.748,E2 -16379.748} C_VEL
LIN {X 0,Y 308.658,Z 461.466,A -85,B 0,C 180,E1 -16380.652,E2 -16380.652} C_VEL
LIN {X 0,Y 307.133,Z 470.811,A -85,B 0,C 180,E1 -16381.804,E2 -16381.804} C_VEL
LIN {X 0,Y 305.71,Z 478.531,A -85,B 0,C 180,E1 -16382.966,E2 -16382.966} C_VEL
LIN {X 0,Y 304.003,Z 487.038,A -85,B 0,C 180,E1 -16384.535,E2 -16384.535} C_VEL
LIN {X 0,Y 302.24,Z 494.649,A -85,B 0,C 180,E1 -16386.342,E2 -16386.342} C_VEL
LIN {X 0,Y 300.859,Z 500.312,A -85,B 0,C 180,E1 -16388.058,E2 -16388.058} C_VEL
LIN {X 0,Y 299.65,Z 505.11,A -85,B 0,C 180,E1 -16389.93,E2 -16389.93} C_VEL
LIN {X 0,Y 298.743,Z 508.268,A -85,B 0,C 180,E1 -16391.536,E2 -16391.536} C_VEL
LIN {X 0,Y 298.44,Z 509.449,A -85,B 0,C 180,E1 -16392.237,E2 -16392.237} C_VEL
LIN {X 0,Y 297.578,Z 511.961,A -85,B 0,C 180,E1 -16394.474,E2 -16394.474} C_VEL
LIN {X 0,Y 297.048,Z 512.984,A -85,B 0,C 180,E1 -16396.495,E2 -16396.495} C_VEL
LIN {X 0,Y 296.802,Z 513.089,A -85,B 0,C 180,E1 -16397.929,E2 -16397.929} C_VEL
LIN {X 0,Y 296.644,Z 512.571,A -85,B 0,C 180,E1 -16399.372,E2 -16399.372} C_VEL
LIN {X 0,Y 296.563,Z 511.41,A -85,B 0,C 180,E1 -16400.823,E2 -16400.823} C_VEL
LIN {X 0,Y 296.715,Z 508.577,A -85,B 0,C 180,E1 -16403.045,E2 -16403.045} C_VEL
LIN {X 0,Y 296.996,Z 504.203,A -85,B 0,C 180,E1 -16405.211,E2 -16405.211} C_VEL
LIN {X 0,Y 297.339,Z 499.182,A -85,B 0,C 180,E1 -16407.066,E2 -16407.066} C_VEL
LIN {X 0,Y 297.746,Z 493.602,A -85,B 0,C 180,E1 -16408.701,E2 -16408.701} C_VEL
LIN {X 0,Y 298.205,Z 487.993,A -85,B 0,C 180,E1 -16410.055,E2 -16410.055} C_VEL
LIN {X 0,Y 298.828,Z 480.725,A -85,B 0,C 180,E1 -16411.513,E2 -16411.513} C_VEL
LIN {X 0,Y 299.572,Z 471.286,A -85,B 0,C 180,E1 -16413.056,E2 -16413.056} C_VEL
LIN {X 0,Y 300.346,Z 461.186,A -85,B 0,C 180,E1 -16414.338,E2 -16414.338} C_VEL
LIN {X 0,Y 300.89,Z 452.246,A -85,B 0,C 180,E1 -16415.256,E2 -16415.256} C_VEL
LIN {X 0,Y 301.462,Z 443.714,A -85,B 0,C 180,E1 -16415.959,E2 -16415.959} C_VEL
LIN {X 0,Y 301.948,Z 433.419,A -85,B 0,C 180,E1 -16416.616,E2 -16416.616} C_VEL
LIN {X 0,Y 302.361,Z 421.301,A -85,B 0,C 180,E1 -16417.156,E2 -16417.156} C_VEL
LIN {X 0,Y 303.856,Z 368.389,A -85,B 0,C 180,E1 -16418.845,E2 -16418.845} C_VEL
LIN {X 0,Y 300.479,Z 339.964,A -85,B 0,C 180,E1 -16419.977,E2 -16419.977} C_VEL
LIN {X 0,Y 302.01,Z 324.078,A -85,B 0,C 180,E1 -16424.278,E2 -16424.278} C_VEL
LIN {X 0,Y 301.808,Z 320.4,A -85,B 0,C 180,E1 -16425.329,E2 -16425.329} C_VEL
LIN {X 0,Y 299.651,Z 309.426,A -85,B 0,C 180,E1 -16428.637,E2 -16428.637} C_VEL
LIN {X 0,Y 298.419,Z 303.313,A -85,B 0,C 180,E1 -16430.593,E2 -16430.593} C_VEL
LIN {X 0,Y 298.403,Z 303.314,A -85,B 0,C 180,E1 -16433.929,E2 -16433.929} C_VEL
LIN {X 0,Y 298.393,Z 303.313,A -85,B 0,C 180,E1 -16437.2,E2 -16437.2} C_VEL
LIN {X 0,Y 298.366,Z 303.317,A -85,B 0,C 180,E1 -16440.639,E2 -16440.639} C_VEL
LIN {X 0,Y 298.415,Z 303.31,A -85,B 0,C 180,E1 -16444.917,E2 -16444.917} C_VEL
LIN {X 0,Y 298.396,Z 303.313,A -85,B 0,C 180,E1 -16447.861,E2 -16447.861} C_VEL
LIN {X 0,Y 298.468,Z 303.308,A -85,B 0,C 180,E1 -16450.751,E2 -16450.751} C_VEL
LIN {X 0,Y 298.592,Z 303.291,A -85,B 0,C 180,E1 -16454.993,E2 -16454.993} C_VEL
LIN {X 0,Y 298.588,Z 303.294,A -85,B 0,C 180,E1 -16459.145,E2 -16459.145} C_VEL
LIN {X 0,Y 298.702,Z 303.274,A -85,B 0,C 180,E1 -16461.882,E2 -16461.882} C_VEL
LIN {X 0,Y 298.629,Z 303.282,A -85,B 0,C 180,E1 -16464.596,E2 -16464.596} C_VEL
LIN {X 0,Y 298.906,Z 303.248,A -85,B 0,C 180,E1 -16468.65,E2 -16468.65} C_VEL
LIN {X 0,Y 298.905,Z 303.25,A -85,B 0,C 180,E1 -16471.344,E2 -16471.344} C_VEL
LIN {X 0,Y 298.735,Z 303.27,A -85,B 0,C 180,E1 -16476.752,E2 -16476.752} C_VEL
LIN {X 0,Y 298.626,Z 303.283,A -85,B 0,C 180,E1 -16479.478,E2 -16479.478} C_VEL
LIN {X 0,Y 298.544,Z 303.293,A -85,B 0,C 180,E1 -16483.612,E2 -16483.612} C_VEL
LIN {X 0,Y 298.482,Z 303.304,A -85,B 0,C 180,E1 -16486.408,E2 -16486.408} C_VEL
LIN {X 0,Y 298.441,Z 303.306,A -85,B 0,C 180,E1 -16489.614,E2 -16489.614} C_VEL
LIN {X 0,Y 298.413,Z 303.311,A -85,B 0,C 180,E1 -16493.596,E2 -16493.596} C_VEL
LIN {X 0,Y 298.399,Z 303.312,A -85,B 0,C 180,E1 -16496.577,E2 -16496.577} C_VEL
LIN {X 0,Y 298.381,Z 303.317,A -85,B 0,C 180,E1 -16499.639,E2 -16499.639} C_VEL
LIN {X 0,Y 298.379,Z 303.314,A -85,B 0,C 180,E1 -16502.795,E2 -16502.795} C_VEL
LIN {X 0,Y 298.413,Z 303.31,A -85,B 0,C 180,E1 -16506.798,E2 -16506.798} C_VEL
LIN {X 0,Y 298.365,Z 303.315,A -85,B 0,C 180,E1 -16511.082,E2 -16511.082} C_VEL
LIN {X 0,Y 298.378,Z 303.314,A -85,B 0,C 180,E1 -16513.098,E2 -16513.098} C_VEL
LIN {X 0,Y 298.349,Z 303.319,A -85,B 0,C 180,E1 -16516.91,E2 -16516.91} C_VEL
LIN {X 0,Y 298.369,Z 303.318,A -85,B 0,C 180,E1 -16521.003,E2 -16521.003} C_VEL
LIN {X 0,Y 298.374,Z 303.315,A -85,B 0,C 180,E1 -16523.923,E2 -16523.923} C_VEL
LIN {X 0,Y 298.362,Z 303.32,A -85,B 0,C 180,E1 -16527.195,E2 -16527.195} C_VEL
LIN {X 0,Y 298.397,Z 303.313,A -85,B 0,C 180,E1 -16530.611,E2 -16530.611} C_VEL
LIN {X 0,Y 298.42,Z 303.31,A -85,B 0,C 180,E1 -16533.976,E2 -16533.976} C_VEL
LIN {X 0,Y 298.367,Z 303.319,A -85,B 0,C 180,E1 -16537.859,E2 -16537.859} C_VEL
LIN {X 0,Y 298.376,Z 303.314,A -85,B 0,C 180,E1 -16539.829,E2 -16539.829} C_VEL
LIN {X 0,Y 297.734,Z 303.395,A -85,B 0,C 180,E1 -16540.956,E2 -16540.956} C_VEL
LIN {X 0,Y 294.904,Z 303.747,A -85,B 0,C 180,E1 -16542.791,E2 -16542.791} C_VEL
LIN {X 0,Y 292.513,Z 304.047,A -85,B 0,C 180,E1 -16544.28,E2 -16544.28} C_VEL
LIN {X 0,Y 291.52,Z 304.169,A -85,B 0,C 180,E1 -16545.434,E2 -16545.434} C_VEL
LIN {X 0,Y 291.458,Z 304.178,A -85,B 0,C 180,E1 -16545.824,E2 -16545.824} C_VEL
LIN {X 0,Y 291.53,Z 304.173,A -85,B 0,C 180,E1 -16550.284,E2 -16550.284} C_VEL
LIN {X 0,Y 291.686,Z 304.148,A -85,B 0,C 180,E1 -16553.08,E2 -16553.08} C_VEL
LIN {X 0,Y 291.757,Z 304.14,A -85,B 0,C 180,E1 -16557.238,E2 -16557.238} C_VEL
LIN {X 0,Y 291.904,Z 304.12,A -85,B 0,C 180,E1 -16559.999,E2 -16559.999} C_VEL
LIN {X 0,Y 291.742,Z 304.143,A -85,B 0,C 180,E1 -16562.761,E2 -16562.761} C_VEL
LIN {X 0,Y 291.685,Z 304.15,A -85,B 0,C 180,E1 -16566.919,E2 -16566.919} C_VEL
LIN {X 0,Y 291.528,Z 304.17,A -85,B 0,C 180,E1 -16569.715,E2 -16569.715} C_VEL
LIN {X 0,Y 291.473,Z 304.178,A -85,B 0,C 180,E1 -16573.952,E2 -16573.952} C_VEL
LIN {X 0,Y 291.421,Z 304.183,A -85,B 0,C 180,E1 -16578.27,E2 -16578.27} C_VEL
LIN {X 0,Y 291.322,Z 304.192,A -85,B 0,C 180,E1 -16581.214,E2 -16581.214} C_VEL
LIN {X 0,Y 291.339,Z 304.196,A -85,B 0,C 180,E1 -16584.21,E2 -16584.21} C_VEL
LIN {X 0,Y 291.363,Z 304.188,A -85,B 0,C 180,E1 -16587.277,E2 -16587.277} C_VEL
LIN {X 0,Y 291.285,Z 304.2,A -85,B 0,C 180,E1 -16590.442,E2 -16590.442} C_VEL
LIN {X 0,Y 291.307,Z 304.195,A -85,B 0,C 180,E1 -16593.702,E2 -16593.702} C_VEL
LIN {X 0,Y 291.337,Z 304.195,A -85,B 0,C 180,E1 -16597.256,E2 -16597.256} C_VEL
LIN {X 0,Y 291.297,Z 304.198,A -85,B 0,C 180,E1 -16600.648,E2 -16600.648} C_VEL
LIN {X 0,Y 291.262,Z 304.201,A -85,B 0,C 180,E1 -16604.406,E2 -16604.406} C_VEL
LIN {X 0,Y 291.299,Z 304.197,A -85,B 0,C 180,E1 -16608.409,E2 -16608.409} C_VEL
LIN {X 0,Y 291.314,Z 304.195,A -85,B 0,C 180,E1 -16611.16,E2 -16611.16} C_VEL
LIN {X 0,Y 291.333,Z 304.193,A -85,B 0,C 180,E1 -16614.63,E2 -16614.63} C_VEL
LIN {X 0,Y 291.409,Z 304.279,A -85,B 0,C 180,E1 -16616.217,E2 -16616.217} C_VEL
LIN {X 0,Y 294.383,Z 317.729,A -85,B 0,C 180,E1 -16619.917,E2 -16619.917} C_VEL
LIN {X 0,Y 296.996,Z 330.572,A -85,B 0,C 180,E1 -16623.287,E2 -16623.287} C_VEL
LIN {X 0,Y 296.118,Z 338.172,A -85,B 0,C 180,E1 -16625.091,E2 -16625.091} C_VEL
LIN {X 0,Y 295.231,Z 344.133,A -85,B 0,C 180,E1 -16626.492,E2 -16626.492} C_VEL
LIN {X 0,Y 297.993,Z 373.961,A -85,B 0,C 180,E1 -16627.548,E2 -16627.548} C_VEL
LIN {X 0,Y 298.108,Z 380.004,A -85,B 0,C 180,E1 -16627.739,E2 -16627.739} C_VEL
LIN {X 0,Y 296.305,Z 446.57,A -85,B 0,C 180,E1 -16629.708,E2 -16629.708} C_VEL
LIN {X 0,Y 295.808,Z 456.734,A -85,B 0,C 180,E1 -16630.171,E2 -16630.171} C_VEL
LIN {X 0,Y 295.234,Z 465.612,A -85,B 0,C 180,E1 -16630.718,E2 -16630.718} C_VEL
LIN {X 0,Y 294.552,Z 474.302,A -85,B 0,C 180,E1 -16631.395,E2 -16631.395} C_VEL
LIN {X 0,Y 293.727,Z 484.679,A -85,B 0,C 180,E1 -16632.422,E2 -16632.422} C_VEL
LIN {X 0,Y 292.947,Z 493.704,A -85,B 0,C 180,E1 -16633.526,E2 -16633.526} C_VEL
LIN {X 0,Y 292.052,Z 502.525,A -85,B 0,C 180,E1 -16634.834,E2 -16634.834} C_VEL
LIN {X 0,Y 291.426,Z 509.453,A -85,B 0,C 180,E1 -16636.049,E2 -16636.049} C_VEL
LIN {X 0,Y 290.893,Z 516.221,A -85,B 0,C 180,E1 -16637.445,E2 -16637.445} C_VEL
LIN {X 0,Y 290.317,Z 523.225,A -85,B 0,C 180,E1 -16639.19,E2 -16639.19} C_VEL
LIN {X 0,Y 289.962,Z 529.01,A -85,B 0,C 180,E1 -16640.939,E2 -16640.939} C_VEL
LIN {X 0,Y 289.814,Z 532.92,A -85,B 0,C 180,E1 -16642.339,E2 -16642.339} C_VEL
LIN {X 0,Y 289.703,Z 537.575,A -85,B 0,C 180,E1 -16644.435,E2 -16644.435} C_VEL
LIN {X 0,Y 289.72,Z 539.923,A -85,B 0,C 180,E1 -16645.83,E2 -16645.83} C_VEL
LIN {X 0,Y 289.756,Z 543.294,A -85,B 0,C 180,E1 -16648.613,E2 -16648.613} C_VEL
LIN {X 0,Y 289.882,Z 544.212,A -85,B 0,C 180,E1 -16650.003,E2 -16650.003} C_VEL
LIN {X 0,Y 289.543,Z 544.796,A -85,B 0,C 180,E1 -16652.785,E2 -16652.785} C_VEL
LIN {X 0,Y 289.507,Z 544.353,A -85,B 0,C 180,E1 -16654.179,E2 -16654.179} C_VEL
LIN {X 0,Y 289.573,Z 542.354,A -85,B 0,C 180,E1 -16656.972,E2 -16656.972} C_VEL
LIN {X 0,Y 289.954,Z 539.646,A -85,B 0,C 180,E1 -16659.067,E2 -16659.067} C_VEL
LIN {X 0,Y 290.566,Z 535.873,A -85,B 0,C 180,E1 -16661.159,E2 -16661.159} C_VEL
LIN {X 0,Y 291.575,Z 530.965,A -85,B 0,C 180,E1 -16663.239,E2 -16663.239} C_VEL
LIN {X 0,Y 293.005,Z 524.75,A -85,B 0,C 180,E1 -16665.3,E2 -16665.3} C_VEL
LIN {X 0,Y 294.332,Z 518.31,A -85,B 0,C 180,E1 -16667.046,E2 -16667.046} C_VEL
LIN {X 0,Y 296.033,Z 510.865,A -85,B 0,C 180,E1 -16668.694,E2 -16668.694} C_VEL
LIN {X 0,Y 297.912,Z 502.646,A -85,B 0,C 180,E1 -16670.184,E2 -16670.184} C_VEL
LIN {X 0,Y 299.46,Z 495.185,A -85,B 0,C 180,E1 -16671.332,E2 -16671.332} C_VEL
LIN {X 0,Y 301.238,Z 486.332,A -85,B 0,C 180,E1 -16672.46,E2 -16672.46} C_VEL
LIN {X 0,Y 302.843,Z 477.208,A -85,B 0,C 180,E1 -16673.417,E2 -16673.417} C_VEL
LIN {X 0,Y 304.355,Z 466.835,A -85,B 0,C 180,E1 -16674.288,E2 -16674.288} C_VEL
LIN {X 0,Y 305.722,Z 456.485,A -85,B 0,C 180,E1 -16674.942,E2 -16674.942} C_VEL
LIN {X 0,Y 306.765,Z 445.734,A -85,B 0,C 180,E1 -16675.44,E2 -16675.44} C_VEL
LIN {X 0,Y 308.022,Z 423.965,A -85,B 0,C 180,E1 -16676.138,E2 -16676.138} C_VEL
LIN {X 0,Y 310.508,Z 378.995,A -85,B 0,C 180,E1 -16677.548,E2 -16677.548} C_VEL
LIN {X 0,Y 308.903,Z 364.422,A -85,B 0,C 180,E1 -16678.387,E2 -16678.387} C_VEL
LIN {X 0,Y 306.02,Z 348.417,A -85,B 0,C 180,E1 -16679.535,E2 -16679.535} C_VEL
LIN {X 0,Y 304.846,Z 345.524,A -85,B 0,C 180,E1 -16679.866,E2 -16679.866} C_VEL
LIN {X 0,Y 303.525,Z 342.508,A -85,B 0,C 180,E1 -16680.239,E2 -16680.239} C_VEL
LIN {X 0,Y 301.673,Z 333.643,A -85,B 0,C 180,E1 -16683,E2 -16683} C_VEL
LIN {X 0,Y 299.385,Z 325.4,A -85,B 0,C 180,E1 -16685.934,E2 -16685.934} C_VEL
LIN {X 0,Y 296.712,Z 317.418,A -85,B 0,C 180,E1 -16689.273,E2 -16689.273} C_VEL
LIN {X 0,Y 294.383,Z 311.565,A -85,B 0,C 180,E1 -16692.262,E2 -16692.262} C_VEL
LIN {X 0,Y 292.523,Z 307.367,A -85,B 0,C 180,E1 -16694.89,E2 -16694.89} C_VEL
LIN {X 0,Y 291.348,Z 304.192,A -85,B 0,C 180,E1 -16697.202,E2 -16697.202} C_VEL
LIN {X 0,Y 291.363,Z 304.192,A -85,B 0,C 180,E1 -16701.161,E2 -16701.161} C_VEL
LIN {X 0,Y 291.356,Z 304.182,A -85,B 0,C 180,E1 -16704.626,E2 -16704.626} C_VEL
LIN {X 0,Y 291.359,Z 304.183,A -85,B 0,C 180,E1 -16707.95,E2 -16707.95} C_VEL
LIN {X 0,Y 291.367,Z 304.183,A -85,B 0,C 180,E1 -16711.158,E2 -16711.158} C_VEL
LIN {X 0,Y 291.399,Z 304.18,A -85,B 0,C 180,E1 -16714.271,E2 -16714.271} C_VEL
LIN {X 0,Y 291.376,Z 304.296,A -85,B 0,C 180,E1 -16717.187,E2 -16717.187} C_VEL
LIN {X 0,Y 293.901,Z 310.172,A -85,B 0,C 180,E1 -16721.167,E2 -16721.167} C_VEL
LIN {X 0,Y 296.09,Z 315.259,A -85,B 0,C 180,E1 -16723.887,E2 -16723.887} C_VEL
LIN {X 0,Y 298.195,Z 320.85,A -85,B 0,C 180,E1 -16726.369,E2 -16726.369} C_VEL
LIN {X 0,Y 300.719,Z 328.351,A -85,B 0,C 180,E1 -16729.225,E2 -16729.225} C_VEL
LIN {X 0,Y 302.703,Z 335.768,A -85,B 0,C 180,E1 -16731.667,E2 -16731.667} C_VEL
LIN {X 0,Y 303.441,Z 339.448,A -85,B 0,C 180,E1 -16732.684,E2 -16732.684} C_VEL
LIN {X 0,Y 304.735,Z 343.12,A -85,B 0,C 180,E1 -16733.097,E2 -16733.097} C_VEL
LIN {X 0,Y 308.254,Z 361.735,A -85,B 0,C 180,E1 -16734.588,E2 -16734.588} C_VEL
LIN {X 0,Y 310.196,Z 375.915,A -85,B 0,C 180,E1 -16735.547,E2 -16735.547} C_VEL
LIN {X 0,Y 306.497,Z 429.274,A -85,B 0,C 180,E1 -16737.495,E2 -16737.495} C_VEL
LIN {X 0,Y 305.39,Z 440.736,A -85,B 0,C 180,E1 -16738.105,E2 -16738.105} C_VEL
LIN {X 0,Y 304.031,Z 452.133,A -85,B 0,C 180,E1 -16738.982,E2 -16738.982} C_VEL
LIN {X 0,Y 302.534,Z 462.208,A -85,B 0,C 180,E1 -16740.001,E2 -16740.001} C_VEL
LIN {X 0,Y 300.896,Z 471.474,A -85,B 0,C 180,E1 -16741.172,E2 -16741.172} C_VEL
LIN {X 0,Y 299.164,Z 480.134,A -85,B 0,C 180,E1 -16742.525,E2 -16742.525} C_VEL
LIN {X 0,Y 297.003,Z 489.69,A -85,B 0,C 180,E1 -16744.442,E2 -16744.442} C_VEL
LIN {X 0,Y 295.685,Z 495.137,A -85,B 0,C 180,E1 -16745.798,E2 -16745.798} C_VEL
LIN {X 0,Y 294.181,Z 500.809,A -85,B 0,C 180,E1 -16747.551,E2 -16747.551} C_VEL
LIN {X 0,Y 292.759,Z 506.059,A -85,B 0,C 180,E1 -16749.675,E2 -16749.675} C_VEL
LIN {X 0,Y 291.566,Z 509.901,A -85,B 0,C 180,E1 -16751.824,E2 -16751.824} C_VEL
LIN {X 0,Y 290.665,Z 512.324,A -85,B 0,C 180,E1 -16753.993,E2 -16753.993} C_VEL
LIN {X 0,Y 290.235,Z 513.237,A -85,B 0,C 180,E1 -16755.449,E2 -16755.449} C_VEL
LIN {X 0,Y 289.87,Z 513.526,A -85,B 0,C 180,E1 -16756.915,E2 -16756.915} C_VEL
LIN {X 0,Y 289.615,Z 513.108,A -85,B 0,C 180,E1 -16758.852,E2 -16758.852} C_VEL
LIN {X 0,Y 289.486,Z 511.099,A -85,B 0,C 180,E1 -16761.357,E2 -16761.357} C_VEL
LIN {X 0,Y 289.607,Z 509.086,A -85,B 0,C 180,E1 -16762.848,E2 -16762.848} C_VEL
LIN {X 0,Y 289.894,Z 504.676,A -85,B 0,C 180,E1 -16765.105,E2 -16765.105} C_VEL
LIN {X 0,Y 290.195,Z 500.322,A -85,B 0,C 180,E1 -16766.79,E2 -16766.79} C_VEL
LIN {X 0,Y 290.524,Z 496.073,A -85,B 0,C 180,E1 -16768.147,E2 -16768.147} C_VEL
LIN {X 0,Y 290.944,Z 490.62,A -85,B 0,C 180,E1 -16769.591,E2 -16769.591} C_VEL
LIN {X 0,Y 291.567,Z 483.099,A -85,B 0,C 180,E1 -16771.215,E2 -16771.215} C_VEL
LIN {X 0,Y 292.146,Z 476.094,A -85,B 0,C 180,E1 -16772.47,E2 -16772.47} C_VEL
LIN {X 0,Y 292.817,Z 467.736,A -85,B 0,C 180,E1 -16773.714,E2 -16773.714} C_VEL
LIN {X 0,Y 293.521,Z 458.234,A -85,B 0,C 180,E1 -16774.867,E2 -16774.867} C_VEL
LIN {X 0,Y 294.3,Z 447.232,A -85,B 0,C 180,E1 -16775.918,E2 -16775.918} C_VEL
LIN {X 0,Y 294.849,Z 435.386,A -85,B 0,C 180,E1 -16776.737,E2 -16776.737} C_VEL
LIN {X 0,Y 295.294,Z 424.69,A -85,B 0,C 180,E1 -16777.259,E2 -16777.259} C_VEL
LIN {X 0,Y 296.918,Z 368.971,A -85,B 0,C 180,E1 -16779.114,E2 -16779.114} C_VEL
LIN {X 0,Y 293.519,Z 340.099,A -85,B 0,C 180,E1 -16780.278,E2 -16780.278} C_VEL
LIN {X 0,Y 295.016,Z 325.246,A -85,B 0,C 180,E1 -16784.386,E2 -16784.386} C_VEL
LIN {X 0,Y 294.993,Z 322.508,A -85,B 0,C 180,E1 -16785.171,E2 -16785.171} C_VEL
LIN {X 0,Y 293.094,Z 312.589,A -85,B 0,C 180,E1 -16788.204,E2 -16788.204} C_VEL
LIN {X 0,Y 291.383,Z 304.189,A -85,B 0,C 180,E1 -16790.9,E2 -16790.9} C_VEL
LIN {X 0,Y 291.355,Z 304.189,A -85,B 0,C 180,E1 -16794.626,E2 -16794.626} C_VEL
LIN {X 0,Y 291.367,Z 304.193,A -85,B 0,C 180,E1 -16797.95,E2 -16797.95} C_VEL
LIN {X 0,Y 291.317,Z 304.194,A -85,B 0,C 180,E1 -16801.151,E2 -16801.151} C_VEL
LIN {X 0,Y 291.345,Z 304.196,A -85,B 0,C 180,E1 -16804.265,E2 -16804.265} C_VEL
LIN {X 0,Y 291.354,Z 304.189,A -85,B 0,C 180,E1 -16807.297,E2 -16807.297} C_VEL
LIN {X 0,Y 291.392,Z 304.187,A -85,B 0,C 180,E1 -16810.265,E2 -16810.265} C_VEL
LIN {X 0,Y 291.503,Z 304.174,A -85,B 0,C 180,E1 -16814.664,E2 -16814.664} C_VEL
LIN {X 0,Y 291.534,Z 304.17,A -85,B 0,C 180,E1 -16818.879,E2 -16818.879} C_VEL
LIN {X 0,Y 291.656,Z 304.153,A -85,B 0,C 180,E1 -16821.685,E2 -16821.685} C_VEL
LIN {X 0,Y 291.6,Z 304.158,A -85,B 0,C 180,E1 -16824.465,E2 -16824.465} C_VEL
LIN {X 0,Y 291.873,Z 304.124,A -85,B 0,C 180,E1 -16828.618,E2 -16828.618} C_VEL
LIN {X 0,Y 291.872,Z 304.126,A -85,B 0,C 180,E1 -16831.377,E2 -16831.377} C_VEL
LIN {X 0,Y 291.687,Z 304.148,A -85,B 0,C 180,E1 -16836.916,E2 -16836.916} C_VEL
LIN {X 0,Y 291.569,Z 304.163,A -85,B 0,C 180,E1 -16839.71,E2 -16839.71} C_VEL
LIN {X 0,Y 291.514,Z 304.169,A -85,B 0,C 180,E1 -16843.946,E2 -16843.946} C_VEL
LIN {X 0,Y 291.426,Z 304.185,A -85,B 0,C 180,E1 -16846.817,E2 -16846.817} C_VEL
LIN {X 0,Y 291.387,Z 304.185,A -85,B 0,C 180,E1 -16849.837,E2 -16849.837} C_VEL
LIN {X 0,Y 291.352,Z 304.189,A -85,B 0,C 180,E1 -16854.204,E2 -16854.204} C_VEL
LIN {X 0,Y 291.344,Z 304.196,A -85,B 0,C 180,E1 -16857.273,E2 -16857.273} C_VEL
LIN {X 0,Y 291.306,Z 304.194,A -85,B 0,C 180,E1 -16860.434,E2 -16860.434} C_VEL
LIN {X 0,Y 291.329,Z 304.198,A -85,B 0,C 180,E1 -16863.693,E2 -16863.693} C_VEL
LIN {X 0,Y 291.344,Z 304.191,A -85,B 0,C 180,E1 -16867.244,E2 -16867.244} C_VEL
LIN {X 0,Y 291.311,Z 304.195,A -85,B 0,C 180,E1 -16870.638,E2 -16870.638} C_VEL
LIN {X 0,Y 291.269,Z 304.204,A -85,B 0,C 180,E1 -16874.396,E2 -16874.396} C_VEL
LIN {X 0,Y 291.291,Z 304.201,A -85,B 0,C 180,E1 -16878.401,E2 -16878.401} C_VEL
LIN {X 0,Y 291.318,Z 304.195,A -85,B 0,C 180,E1 -16881.152,E2 -16881.152} C_VEL
LIN {X 0,Y 291.325,Z 304.196,A -85,B 0,C 180,E1 -16884.62,E2 -16884.62} C_VEL
LIN {X 0,Y 291.338,Z 304.19,A -85,B 0,C 180,E1 -16887.946,E2 -16887.946} C_VEL
LIN {X 0,Y 291.343,Z 304.195,A -85,B 0,C 180,E1 -16891.153,E2 -16891.153} C_VEL
LIN {X 0,Y 291.374,Z 304.186,A -85,B 0,C 180,E1 -16894.267,E2 -16894.267} C_VEL
LIN {X 0,Y 291.33,Z 304.194,A -85,B 0,C 180,E1 -16897.295,E2 -16897.295} C_VEL
LIN {X 0,Y 291.349,Z 304.191,A -85,B 0,C 180,E1 -16900.262,E2 -16900.262} C_VEL
LIN {X 0,Y 291.457,Z 304.176,A -85,B 0,C 180,E1 -16904.663,E2 -16904.663} C_VEL
LIN {X 0,Y 291.458,Z 304.178,A -85,B 0,C 180,E1 -16905.824,E2 -16905.824} C_VEL
LIN {X 0,Y 290.849,Z 304.261,A -85,B 0,C 180,E1 -16906.977,E2 -16906.977} C_VEL
LIN {X 0,Y 288.06,Z 304.609,A -85,B 0,C 180,E1 -16908.857,E2 -16908.857} C_VEL
LIN {X 0,Y 285.674,Z 304.902,A -85,B 0,C 180,E1 -16910.383,E2 -16910.383} C_VEL
LIN {X 0,Y 284.66,Z 305.023,A -85,B 0,C 180,E1 -16911.564,E2 -16911.564} C_VEL
LIN {X 0,Y 284.585,Z 305.03,A -85,B 0,C 180,E1 -16911.964,E2 -16911.964} C_VEL
LIN {X 0,Y 284.47,Z 305.046,A -85,B 0,C 180,E1 -16915.749,E2 -16915.749} C_VEL
LIN {X 0,Y 284.813,Z 305.008,A -85,B 0,C 180,E1 -16918.585,E2 -16918.585} C_VEL
LIN {X 0,Y 284.809,Z 305.005,A -85,B 0,C 180,E1 -16921.413,E2 -16921.413} C_VEL
LIN {X 0,Y 284.636,Z 305.03,A -85,B 0,C 180,E1 -16927.091,E2 -16927.091} C_VEL
LIN {X 0,Y 284.474,Z 305.047,A -85,B 0,C 180,E1 -16929.958,E2 -16929.958} C_VEL
LIN {X 0,Y 284.425,Z 305.053,A -85,B 0,C 180,E1 -16934.305,E2 -16934.305} C_VEL
LIN {X 0,Y 284.355,Z 305.061,A -85,B 0,C 180,E1 -16938.741,E2 -16938.741} C_VEL
LIN {X 0,Y 284.277,Z 305.072,A -85,B 0,C 180,E1 -16941.766,E2 -16941.766} C_VEL
LIN {X 0,Y 284.293,Z 305.07,A -85,B 0,C 180,E1 -16944.85,E2 -16944.85} C_VEL
LIN {X 0,Y 284.273,Z 305.072,A -85,B 0,C 180,E1 -16948.016,E2 -16948.016} C_VEL
LIN {X 0,Y 284.249,Z 305.075,A -85,B 0,C 180,E1 -16951.279,E2 -16951.279} C_VEL
LIN {X 0,Y 284.302,Z 305.069,A -85,B 0,C 180,E1 -16955.35,E2 -16955.35} C_VEL
LIN {X 0,Y 284.274,Z 305.072,A -85,B 0,C 180,E1 -16958.174,E2 -16958.174} C_VEL
LIN {X 0,Y 284.222,Z 305.078,A -85,B 0,C 180,E1 -16962.124,E2 -16962.124} C_VEL
LIN {X 0,Y 284.229,Z 305.078,A -85,B 0,C 180,E1 -16966.194,E2 -16966.194} C_VEL
LIN {X 0,Y 284.282,Z 305.074,A -85,B 0,C 180,E1 -16970.029,E2 -16970.029} C_VEL
LIN {X 0,Y 284.297,Z 305.072,A -85,B 0,C 180,E1 -16973.617,E2 -16973.617} C_VEL
LIN {X 0,Y 284.318,Z 305.151,A -85,B 0,C 180,E1 -16975.836,E2 -16975.836} C_VEL
LIN {X 0,Y 287.22,Z 318.11,A -85,B 0,C 180,E1 -16979.494,E2 -16979.494} C_VEL
LIN {X 0,Y 289.891,Z 331.029,A -85,B 0,C 180,E1 -16982.969,E2 -16982.969} C_VEL
LIN {X 0,Y 290.068,Z 332.602,A -85,B 0,C 180,E1 -16983.376,E2 -16983.376} C_VEL
LIN {X 0,Y 288.315,Z 344.314,A -85,B 0,C 180,E1 -16986.156,E2 -16986.156} C_VEL
LIN {X 0,Y 291.153,Z 375.287,A -85,B 0,C 180,E1 -16987.286,E2 -16987.286} C_VEL
LIN {X 0,Y 289.879,Z 427.771,A -85,B 0,C 180,E1 -16988.866,E2 -16988.866} C_VEL
LIN {X 0,Y 289.261,Z 447.954,A -85,B 0,C 180,E1 -16989.517,E2 -16989.517} C_VEL
LIN {X 0,Y 288.535,Z 460.658,A -85,B 0,C 180,E1 -16990.16,E2 -16990.16} C_VEL
LIN {X 0,Y 287.584,Z 473.273,A -85,B 0,C 180,E1 -16991.112,E2 -16991.112} C_VEL
LIN {X 0,Y 286.764,Z 483.775,A -85,B 0,C 180,E1 -16992.165,E2 -16992.165} C_VEL
LIN {X 0,Y 286.013,Z 492.332,A -85,B 0,C 180,E1 -16993.216,E2 -16993.216} C_VEL
LIN {X 0,Y 285.032,Z 501.773,A -85,B 0,C 180,E1 -16994.634,E2 -16994.634} C_VEL
LIN {X 0,Y 284.328,Z 509.633,A -85,B 0,C 180,E1 -16996.059,E2 -16996.059} C_VEL
LIN {X 0,Y 283.796,Z 516.308,A -85,B 0,C 180,E1 -16997.49,E2 -16997.49} C_VEL
LIN {X 0,Y 283.228,Z 523.226,A -85,B 0,C 180,E1 -16999.278,E2 -16999.278} C_VEL
LIN {X 0,Y 282.933,Z 527.95,A -85,B 0,C 180,E1 -17000.712,E2 -17000.712} C_VEL
LIN {X 0,Y 282.704,Z 533.607,A -85,B 0,C 180,E1 -17002.863,E2 -17002.863} C_VEL
LIN {X 0,Y 282.671,Z 537.954,A -85,B 0,C 180,E1 -17005.011,E2 -17005.011} C_VEL
LIN {X 0,Y 282.577,Z 541.098,A -85,B 0,C 180,E1 -17007.152,E2 -17007.152} C_VEL
LIN {X 0,Y 282.669,Z 542.677,A -85,B 0,C 180,E1 -17008.578,E2 -17008.578} C_VEL
LIN {X 0,Y 282.826,Z 543.63,A -85,B 0,C 180,E1 -17010.003,E2 -17010.003} C_VEL
LIN {X 0,Y 282.467,Z 544.382,A -85,B 0,C 180,E1 -17012.855,E2 -17012.855} C_VEL
LIN {X 0,Y 282.436,Z 543.245,A -85,B 0,C 180,E1 -17015.715,E2 -17015.715} C_VEL
LIN {X 0,Y 282.497,Z 542.122,A -85,B 0,C 180,E1 -17017.148,E2 -17017.148} C_VEL
LIN {X 0,Y 282.905,Z 539.532,A -85,B 0,C 180,E1 -17019.294,E2 -17019.294} C_VEL
LIN {X 0,Y 283.578,Z 535.907,A -85,B 0,C 180,E1 -17021.437,E2 -17021.437} C_VEL
LIN {X 0,Y 284.654,Z 531.153,A -85,B 0,C 180,E1 -17023.567,E2 -17023.567} C_VEL
LIN {X 0,Y 286.168,Z 525.088,A -85,B 0,C 180,E1 -17025.674,E2 -17025.674} C_VEL
LIN {X 0,Y 287.706,Z 518.193,A -85,B 0,C 180,E1 -17027.605,E2 -17027.605} C_VEL
LIN {X 0,Y 289.37,Z 511.578,A -85,B 0,C 180,E1 -17029.141,E2 -17029.141} C_VEL
LIN {X 0,Y 291.561,Z 502.626,A -85,B 0,C 180,E1 -17030.828,E2 -17030.828} C_VEL
LIN {X 0,Y 293.498,Z 494.027,A -85,B 0,C 180,E1 -17032.158,E2 -17032.158} C_VEL
LIN {X 0,Y 295.357,Z 485.01,A -85,B 0,C 180,E1 -17033.303,E2 -17033.303} C_VEL
LIN {X 0,Y 297.01,Z 475.677,A -85,B 0,C 180,E1 -17034.277,E2 -17034.277} C_VEL
LIN {X 0,Y 298.655,Z 464.984,A -85,B 0,C 180,E1 -17035.154,E2 -17035.154} C_VEL
LIN {X 0,Y 299.934,Z 455.767,A -85,B 0,C 180,E1 -17035.736,E2 -17035.736} C_VEL
LIN {X 0,Y 301.011,Z 445.089,A -85,B 0,C 180,E1 -17036.241,E2 -17036.241} C_VEL
LIN {X 0,Y 302.2,Z 426.331,A -85,B 0,C 180,E1 -17036.866,E2 -17036.866} C_VEL
LIN {X 0,Y 304.953,Z 380.401,A -85,B 0,C 180,E1 -17038.331,E2 -17038.331} C_VEL
LIN {X 0,Y 303.518,Z 366.609,A -85,B 0,C 180,E1 -17039.157,E2 -17039.157} C_VEL
LIN {X 0,Y 300.957,Z 351.296,A -85,B 0,C 180,E1 -17040.298,E2 -17040.298} C_VEL
LIN {X 0,Y 296.756,Z 342.427,A -85,B 0,C 180,E1 -17041.508,E2 -17041.508} C_VEL
LIN {X 0,Y 294.76,Z 333.613,A -85,B 0,C 180,E1 -17044.49,E2 -17044.49} C_VEL
LIN {X 0,Y 292.478,Z 325.873,A -85,B 0,C 180,E1 -17047.538,E2 -17047.538} C_VEL
LIN {X 0,Y 290.38,Z 319.872,A -85,B 0,C 180,E1 -17050.327,E2 -17050.327} C_VEL
LIN {X 0,Y 288.435,Z 315.024,A -85,B 0,C 180,E1 -17053.032,E2 -17053.032} C_VEL
LIN {X 0,Y 287.014,Z 311.699,A -85,B 0,C 180,E1 -17055.242,E2 -17055.242} C_VEL
LIN {X 0,Y 285.906,Z 308.798,A -85,B 0,C 180,E1 -17057.512,E2 -17057.512} C_VEL
LIN {X 0,Y 284.322,Z 305.064,A -85,B 0,C 180,E1 -17061.834,E2 -17061.834} C_VEL
LIN {X 0,Y 284.299,Z 305.062,A -85,B 0,C 180,E1 -17065.35,E2 -17065.35} C_VEL
LIN {X 0,Y 284.283,Z 305.064,A -85,B 0,C 180,E1 -17068.725,E2 -17068.725} C_VEL
LIN {X 0,Y 284.387,Z 305.143,A -85,B 0,C 180,E1 -17072.67,E2 -17072.67} C_VEL
LIN {X 0,Y 286.073,Z 308.887,A -85,B 0,C 180,E1 -17076.855,E2 -17076.855} C_VEL
LIN {X 0,Y 288.423,Z 314.386,A -85,B 0,C 180,E1 -17080.796,E2 -17080.796} C_VEL
LIN {X 0,Y 290.711,Z 319.939,A -85,B 0,C 180,E1 -17083.86,E2 -17083.86} C_VEL
LIN {X 0,Y 293.133,Z 326.82,A -85,B 0,C 180,E1 -17086.925,E2 -17086.925} C_VEL
LIN {X 0,Y 295.62,Z 334.88,A -85,B 0,C 180,E1 -17089.947,E2 -17089.947} C_VEL
LIN {X 0,Y 296.809,Z 339.504,A -85,B 0,C 180,E1 -17091.431,E2 -17091.431} C_VEL
LIN {X 0,Y 299.645,Z 345.856,A -85,B 0,C 180,E1 -17092.314,E2 -17092.314} C_VEL
LIN {X 0,Y 302.931,Z 364.119,A -85,B 0,C 180,E1 -17093.835,E2 -17093.835} C_VEL
LIN {X 0,Y 304.626,Z 377.019,A -85,B 0,C 180,E1 -17094.747,E2 -17094.747} C_VEL
LIN {X 0,Y 300.787,Z 429.31,A -85,B 0,C 180,E1 -17096.694,E2 -17096.694} C_VEL
LIN {X 0,Y 299.643,Z 440.661,A -85,B 0,C 180,E1 -17097.312,E2 -17097.312} C_VEL
LIN {X 0,Y 297.974,Z 453.315,A -85,B 0,C 180,E1 -17098.311,E2 -17098.311} C_VEL
LIN {X 0,Y 296.524,Z 462.371,A -85,B 0,C 180,E1 -17099.251,E2 -17099.251} C_VEL
LIN {X 0,Y 295,Z 470.724,A -85,B 0,C 180,E1 -17100.308,E2 -17100.308} C_VEL
LIN {X 0,Y 293.322,Z 478.766,A -85,B 0,C 180,E1 -17101.545,E2 -17101.545} C_VEL
LIN {X 0,Y 291.836,Z 485.301,A -85,B 0,C 180,E1 -17102.761,E2 -17102.761} C_VEL
LIN {X 0,Y 290.206,Z 491.633,A -85,B 0,C 180,E1 -17104.167,E2 -17104.167} C_VEL
LIN {X 0,Y 288.8,Z 496.901,A -85,B 0,C 180,E1 -17105.587,E2 -17105.587} C_VEL
LIN {X 0,Y 287.533,Z 501.315,A -85,B 0,C 180,E1 -17107.021,E2 -17107.021} C_VEL
LIN {X 0,Y 285.999,Z 506.557,A -85,B 0,C 180,E1 -17109.192,E2 -17109.192} C_VEL
LIN {X 0,Y 284.712,Z 510.388,A -85,B 0,C 180,E1 -17111.39,E2 -17111.39} C_VEL
LIN {X 0,Y 284.022,Z 512.087,A -85,B 0,C 180,E1 -17112.869,E2 -17112.869} C_VEL
LIN {X 0,Y 283.354,Z 513.451,A -85,B 0,C 180,E1 -17114.7,E2 -17114.7} C_VEL
LIN {X 0,Y 282.701,Z 513.974,A -85,B 0,C 180,E1 -17117.358,E2 -17117.358} C_VEL
LIN {X 0,Y 282.503,Z 513.365,A -85,B 0,C 180,E1 -17119.038,E2 -17119.038} C_VEL
LIN {X 0,Y 282.389,Z 512.284,A -85,B 0,C 180,E1 -17120.392,E2 -17120.392} C_VEL
LIN {X 0,Y 282.522,Z 508.954,A -85,B 0,C 180,E1 -17123.02,E2 -17123.02} C_VEL
LIN {X 0,Y 282.777,Z 505.115,A -85,B 0,C 180,E1 -17124.994,E2 -17124.994} C_VEL
LIN {X 0,Y 283.094,Z 500.937,A -85,B 0,C 180,E1 -17126.66,E2 -17126.66} C_VEL
LIN {X 0,Y 283.51,Z 495.12,A -85,B 0,C 180,E1 -17128.503,E2 -17128.503} C_VEL
LIN {X 0,Y 283.972,Z 489.408,A -85,B 0,C 180,E1 -17129.983,E2 -17129.983} C_VEL
LIN {X 0,Y 284.458,Z 483.589,A -85,B 0,C 180,E1 -17131.255,E2 -17131.255} C_VEL
LIN {X 0,Y 285.094,Z 476.069,A -85,B 0,C 180,E1 -17132.634,E2 -17132.634} C_VEL
LIN {X 0,Y 285.77,Z 468.166,A -85,B 0,C 180,E1 -17133.837,E2 -17133.837} C_VEL
LIN {X 0,Y 286.471,Z 458.932,A -85,B 0,C 180,E1 -17134.993,E2 -17134.993} C_VEL
LIN {X 0,Y 287.341,Z 446.68,A -85,B 0,C 180,E1 -17136.186,E2 -17136.186} C_VEL
LIN {X 0,Y 287.889,Z 435.131,A -85,B 0,C 180,E1 -17136.993,E2 -17136.993} C_VEL
LIN {X 0,Y 288.311,Z 425.026,A -85,B 0,C 180,E1 -17137.496,E2 -17137.496} C_VEL
LIN {X 0,Y 289.976,Z 369.333,A -85,B 0,C 180,E1 -17139.404,E2 -17139.404} C_VEL
LIN {X 0,Y 286.592,Z 340.088,A -85,B 0,C 180,E1 -17140.634,E2 -17140.634} C_VEL
LIN {X 0,Y 288.017,Z 326.305,A -85,B 0,C 180,E1 -17144.526,E2 -17144.526} C_VEL
LIN {X 0,Y 287.895,Z 323.098,A -85,B 0,C 180,E1 -17145.47,E2 -17145.47} C_VEL
LIN {X 0,Y 285.79,Z 312.323,A -85,B 0,C 180,E1 -17148.849,E2 -17148.849} C_VEL
LIN {X 0,Y 284.323,Z 305.07,A -85,B 0,C 180,E1 -17151.269,E2 -17151.269} C_VEL
LIN {X 0,Y 284.308,Z 305.069,A -85,B 0,C 180,E1 -17155.351,E2 -17155.351} C_VEL
LIN {X 0,Y 284.279,Z 305.071,A -85,B 0,C 180,E1 -17158.724,E2 -17158.724} C_VEL
LIN {X 0,Y 284.262,Z 305.077,A -85,B 0,C 180,E1 -17161.982,E2 -17161.982} C_VEL
LIN {X 0,Y 284.286,Z 305.07,A -85,B 0,C 180,E1 -17165.148,E2 -17165.148} C_VEL
LIN {X 0,Y 284.303,Z 305.071,A -85,B 0,C 180,E1 -17168.234,E2 -17168.234} C_VEL
LIN {X 0,Y 284.335,Z 305.064,A -85,B 0,C 180,E1 -17171.256,E2 -17171.256} C_VEL
LIN {X 0,Y 284.469,Z 305.046,A -85,B 0,C 180,E1 -17175.695,E2 -17175.695} C_VEL
LIN {X 0,Y 284.52,Z 305.041,A -85,B 0,C 180,E1 -17180.041,E2 -17180.041} C_VEL
LIN {X 0,Y 284.646,Z 305.027,A -85,B 0,C 180,E1 -17182.906,E2 -17182.906} C_VEL
LIN {X 0,Y 284.84,Z 305.001,A -85,B 0,C 180,E1 -17188.583,E2 -17188.583} C_VEL
LIN {X 0,Y 284.839,Z 305.003,A -85,B 0,C 180,E1 -17191.411,E2 -17191.411} C_VEL
LIN {X 0,Y 284.643,Z 305.025,A -85,B 0,C 180,E1 -17197.088,E2 -17197.088} C_VEL
LIN {X 0,Y 284.515,Z 305.044,A -85,B 0,C 180,E1 -17199.953,E2 -17199.953} C_VEL
LIN {X 0,Y 284.462,Z 305.05,A -85,B 0,C 180,E1 -17204.299,E2 -17204.299} C_VEL
LIN {X 0,Y 284.33,Z 305.069,A -85,B 0,C 180,E1 -17208.738,E2 -17208.738} C_VEL
LIN {X 0,Y 284.32,Z 305.069,A -85,B 0,C 180,E1 -17213.291,E2 -17213.291} C_VEL
LIN {X 0,Y 284.32,Z 305.07,A -85,B 0,C 180,E1 -17217.141,E2 -17217.141} C_VEL
LIN {X 0,Y 284.284,Z 305.069,A -85,B 0,C 180,E1 -17220.086,E2 -17220.086} C_VEL
LIN {X 0,Y 284.291,Z 305.069,A -85,B 0,C 180,E1 -17222.94,E2 -17222.94} C_VEL
LIN {X 0,Y 284.306,Z 305.068,A -85,B 0,C 180,E1 -17226.382,E2 -17226.382} C_VEL
LIN {X 0,Y 284.287,Z 305.074,A -85,B 0,C 180,E1 -17229.989,E2 -17229.989} C_VEL
LIN {X 0,Y 284.225,Z 305.082,A -85,B 0,C 180,E1 -17234.185,E2 -17234.185} C_VEL
LIN {X 0,Y 284.233,Z 305.078,A -85,B 0,C 180,E1 -17238.116,E2 -17238.116} C_VEL
LIN {X 0,Y 284.276,Z 305.071,A -85,B 0,C 180,E1 -17241.824,E2 -17241.824} C_VEL
LIN {X 0,Y 284.276,Z 305.072,A -85,B 0,C 180,E1 -17245.345,E2 -17245.345} C_VEL
LIN {X 0,Y 284.262,Z 305.074,A -85,B 0,C 180,E1 -17248.721,E2 -17248.721} C_VEL
LIN {X 0,Y 284.358,Z 305.062,A -85,B 0,C 180,E1 -17252.824,E2 -17252.824} C_VEL
LIN {X 0,Y 284.294,Z 305.067,A -85,B 0,C 180,E1 -17256.7,E2 -17256.7} C_VEL
LIN {X 0,Y 284.288,Z 305.071,A -85,B 0,C 180,E1 -17261.253,E2 -17261.253} C_VEL
LIN {X 0,Y 284.421,Z 305.054,A -85,B 0,C 180,E1 -17265.693,E2 -17265.693} C_VEL
LIN {X 0,Y 284.475,Z 305.049,A -85,B 0,C 180,E1 -17270.041,E2 -17270.041} C_VEL
LIN {X 0,Y 284.585,Z 305.03,A -85,B 0,C 180,E1 -17271.964,E2 -17271.964} C_VEL
LIN {X 0,Y 283.932,Z 305.114,A -85,B 0,C 180,E1 -17273.144,E2 -17273.144} C_VEL
LIN {X 0,Y 281.091,Z 305.469,A -85,B 0,C 180,E1 -17275.067,E2 -17275.067} C_VEL
LIN {X 0,Y 278.724,Z 305.767,A -85,B 0,C 180,E1 -17276.628,E2 -17276.628} C_VEL
LIN {X 0,Y 277.779,Z 305.881,A -85,B 0,C 180,E1 -17277.838,E2 -17277.838} C_VEL
LIN {X 0,Y 277.741,Z 305.886,A -85,B 0,C 180,E1 -17278.247,E2 -17278.247} C_VEL
LIN {X 0,Y 277.775,Z 305.881,A -85,B 0,C 180,E1 -17281.449,E2 -17281.449} C_VEL
LIN {X 0,Y 277.59,Z 305.909,A -85,B 0,C 180,E1 -17287.272,E2 -17287.272} C_VEL
LIN {X 0,Y 277.417,Z 305.925,A -85,B 0,C 180,E1 -17290.214,E2 -17290.214} C_VEL
LIN {X 0,Y 277.373,Z 305.931,A -85,B 0,C 180,E1 -17294.677,E2 -17294.677} C_VEL
LIN {X 0,Y 277.3,Z 305.94,A -85,B 0,C 180,E1 -17299.236,E2 -17299.236} C_VEL
LIN {X 0,Y 277.25,Z 305.95,A -85,B 0,C 180,E1 -17304.158,E2 -17304.158} C_VEL
LIN {X 0,Y 277.271,Z 305.943,A -85,B 0,C 180,E1 -17307.501,E2 -17307.501} C_VEL
LIN {X 0,Y 277.213,Z 305.953,A -85,B 0,C 180,E1 -17310.476,E2 -17310.476} C_VEL
LIN {X 0,Y 277.211,Z 305.951,A -85,B 0,C 180,E1 -17313.9,E2 -17313.9} C_VEL
LIN {X 0,Y 277.23,Z 305.951,A -85,B 0,C 180,E1 -17317.474,E2 -17317.474} C_VEL
LIN {X 0,Y 277.171,Z 305.962,A -85,B 0,C 180,E1 -17321.242,E2 -17321.242} C_VEL
LIN {X 0,Y 277.174,Z 305.959,A -85,B 0,C 180,E1 -17325.231,E2 -17325.231} C_VEL
LIN {X 0,Y 277.198,Z 305.957,A -85,B 0,C 180,E1 -17329.517,E2 -17329.517} C_VEL
LIN {X 0,Y 277.231,Z 305.95,A -85,B 0,C 180,E1 -17332.533,E2 -17332.533} C_VEL
LIN {X 0,Y 277.275,Z 306.092,A -85,B 0,C 180,E1 -17335.457,E2 -17335.457} C_VEL
LIN {X 0,Y 280.449,Z 320.273,A -85,B 0,C 180,E1 -17339.563,E2 -17339.563} C_VEL
LIN {X 0,Y 283.003,Z 333.016,A -85,B 0,C 180,E1 -17343.057,E2 -17343.057} C_VEL
LIN {X 0,Y 281.416,Z 343.927,A -85,B 0,C 180,E1 -17345.769,E2 -17345.769} C_VEL
LIN {X 0,Y 283.953,Z 373.511,A -85,B 0,C 180,E1 -17346.898,E2 -17346.898} C_VEL
LIN {X 0,Y 284.337,Z 378.338,A -85,B 0,C 180,E1 -17347.073,E2 -17347.073} C_VEL
LIN {X 0,Y 282.306,Z 446.388,A -85,B 0,C 180,E1 -17349.227,E2 -17349.227} C_VEL
LIN {X 0,Y 281.824,Z 456.385,A -85,B 0,C 180,E1 -17349.714,E2 -17349.714} C_VEL
LIN {X 0,Y 281.208,Z 465.148,A -85,B 0,C 180,E1 -17350.287,E2 -17350.287} C_VEL
LIN {X 0,Y 280.529,Z 473.794,A -85,B 0,C 180,E1 -17350.998,E2 -17350.998} C_VEL
LIN {X 0,Y 279.685,Z 484.13,A -85,B 0,C 180,E1 -17352.077,E2 -17352.077} C_VEL
LIN {X 0,Y 278.917,Z 492.418,A -85,B 0,C 180,E1 -17353.131,E2 -17353.131} C_VEL
LIN {X 0,Y 278.04,Z 500.88,A -85,B 0,C 180,E1 -17354.426,E2 -17354.426} C_VEL
LIN {X 0,Y 277.221,Z 509.694,A -85,B 0,C 180,E1 -17356.068,E2 -17356.068} C_VEL
LIN {X 0,Y 276.679,Z 516.299,A -85,B 0,C 180,E1 -17357.535,E2 -17357.535} C_VEL
LIN {X 0,Y 276.138,Z 523.16,A -85,B 0,C 180,E1 -17359.371,E2 -17359.371} C_VEL
LIN {X 0,Y 275.805,Z 528.811,A -85,B 0,C 180,E1 -17361.209,E2 -17361.209} C_VEL
LIN {X 0,Y 275.653,Z 532.647,A -85,B 0,C 180,E1 -17362.68,E2 -17362.68} C_VEL
LIN {X 0,Y 275.586,Z 536.612,A -85,B 0,C 180,E1 -17364.574,E2 -17364.574} C_VEL
LIN {X 0,Y 275.505,Z 540.402,A -85,B 0,C 180,E1 -17367.079,E2 -17367.079} C_VEL
LIN {X 0,Y 275.587,Z 542.002,A -85,B 0,C 180,E1 -17368.542,E2 -17368.542} C_VEL
LIN {X 0,Y 275.77,Z 543.048,A -85,B 0,C 180,E1 -17370.003,E2 -17370.003} C_VEL
LIN {X 0,Y 275.439,Z 543.708,A -85,B 0,C 180,E1 -17371.465,E2 -17371.465} C_VEL
LIN {X 0,Y 275.391,Z 543.919,A -85,B 0,C 180,E1 -17372.928,E2 -17372.928} C_VEL
LIN {X 0,Y 275.342,Z 542.985,A -85,B 0,C 180,E1 -17375.862,E2 -17375.862} C_VEL
LIN {X 0,Y 275.446,Z 541.871,A -85,B 0,C 180,E1 -17377.332,E2 -17377.332} C_VEL
LIN {X 0,Y 276.078,Z 538.354,A -85,B 0,C 180,E1 -17380.267,E2 -17380.267} C_VEL
LIN {X 0,Y 276.899,Z 534.469,A -85,B 0,C 180,E1 -17382.461,E2 -17382.461} C_VEL
LIN {X 0,Y 278.234,Z 529.425,A -85,B 0,C 180,E1 -17384.633,E2 -17384.633} C_VEL
LIN {X 0,Y 279.612,Z 524.298,A -85,B 0,C 180,E1 -17386.427,E2 -17386.427} C_VEL
LIN {X 0,Y 281.185,Z 518.008,A -85,B 0,C 180,E1 -17388.238,E2 -17388.238} C_VEL
LIN {X 0,Y 283.134,Z 510.672,A -85,B 0,C 180,E1 -17389.957,E2 -17389.957} C_VEL
LIN {X 0,Y 285.183,Z 502.633,A -85,B 0,C 180,E1 -17391.505,E2 -17391.505} C_VEL
LIN {X 0,Y 287.284,Z 494.095,A -85,B 0,C 180,E1 -17392.853,E2 -17392.853} C_VEL
LIN {X 0,Y 289.249,Z 485.258,A -85,B 0,C 180,E1 -17394.016,E2 -17394.016} C_VEL
LIN {X 0,Y 290.989,Z 476.172,A -85,B 0,C 180,E1 -17395.003,E2 -17395.003} C_VEL
LIN {X 0,Y 292.717,Z 465.829,A -85,B 0,C 180,E1 -17395.892,E2 -17395.892} C_VEL
LIN {X 0,Y 294.22,Z 455.536,A -85,B 0,C 180,E1 -17396.56,E2 -17396.56} C_VEL
LIN {X 0,Y 295.368,Z 444.905,A -85,B 0,C 180,E1 -17397.069,E2 -17397.069} C_VEL
LIN {X 0,Y 296.492,Z 428.573,A -85,B 0,C 180,E1 -17397.627,E2 -17397.627} C_VEL
LIN {X 0,Y 299.492,Z 381.095,A -85,B 0,C 180,E1 -17399.196,E2 -17399.196} C_VEL
LIN {X 0,Y 298.082,Z 367.137,A -85,B 0,C 180,E1 -17400.082,E2 -17400.082} C_VEL
LIN {X 0,Y 295.923,Z 354.553,A -85,B 0,C 180,E1 -17401.073,E2 -17401.073} C_VEL
LIN {X 0,Y 291.721,Z 345.821,A -85,B 0,C 180,E1 -17402.371,E2 -17402.371} C_VEL
LIN {X 0,Y 289.94,Z 342.178,A -85,B 0,C 180,E1 -17402.985,E2 -17402.985} C_VEL
LIN {X 0,Y 288.117,Z 334.456,A -85,B 0,C 180,E1 -17405.833,E2 -17405.833} C_VEL
LIN {X 0,Y 285.719,Z 326.724,A -85,B 0,C 180,E1 -17409.213,E2 -17409.213} C_VEL
LIN {X 0,Y 283.783,Z 321.443,A -85,B 0,C 180,E1 -17412.017,E2 -17412.017} C_VEL
LIN {X 0,Y 281.939,Z 316.823,A -85,B 0,C 180,E1 -17415.03,E2 -17415.03} C_VEL
LIN {X 0,Y 280.746,Z 313.759,A -85,B 0,C 180,E1 -17417.477,E2 -17417.477} C_VEL
LIN {X 0,Y 279.333,Z 310.51,A -85,B 0,C 180,E1 -17421.254,E2 -17421.254} C_VEL
LIN {X 0,Y 278.642,Z 309.3,A -85,B 0,C 180,E1 -17423.812,E2 -17423.812} C_VEL
LIN {X 0,Y 278.267,Z 308.829,A -85,B 0,C 180,E1 -17427.97,E2 -17427.97} C_VEL
LIN {X 0,Y 279.046,Z 309.813,A -85,B 0,C 180,E1 -17431.82,E2 -17431.82} C_VEL
LIN {X 0,Y 279.406,Z 310.563,A -85,B 0,C 180,E1 -17433.08,E2 -17433.08} C_VEL
LIN {X 0,Y 280.678,Z 313.44,A -85,B 0,C 180,E1 -17436.383,E2 -17436.383} C_VEL
LIN {X 0,Y 283.081,Z 318.983,A -85,B 0,C 180,E1 -17440.626,E2 -17440.626} C_VEL
LIN {X 0,Y 285.351,Z 324.655,A -85,B 0,C 180,E1 -17443.841,E2 -17443.841} C_VEL
LIN {X 0,Y 287.344,Z 330.589,A -85,B 0,C 180,E1 -17446.565,E2 -17446.565} C_VEL
LIN {X 0,Y 289.299,Z 336.948,A -85,B 0,C 180,E1 -17449.085,E2 -17449.085} C_VEL
LIN {X 0,Y 290.019,Z 339.51,A -85,B 0,C 180,E1 -17449.989,E2 -17449.989} C_VEL
LIN {X 0,Y 294.31,Z 347.972,A -85,B 0,C 180,E1 -17451.383,E2 -17451.383} C_VEL
LIN {X 0,Y 295.217,Z 351.488,A -85,B 0,C 180,E1 -17451.765,E2 -17451.765} C_VEL
LIN {X 0,Y 298.178,Z 369.586,A -85,B 0,C 180,E1 -17453.279,E2 -17453.279} C_VEL
LIN {X 0,Y 299.16,Z 378.415,A -85,B 0,C 180,E1 -17453.909,E2 -17453.909} C_VEL
LIN {X 0,Y 295.09,Z 430.33,A -85,B 0,C 180,E1 -17455.903,E2 -17455.903} C_VEL
LIN {X 0,Y 293.799,Z 442.203,A -85,B 0,C 180,E1 -17456.572,E2 -17456.572} C_VEL
LIN {X 0,Y 292.04,Z 454.46,A -85,B 0,C 180,E1 -17457.587,E2 -17457.587} C_VEL
LIN {X 0,Y 290.411,Z 463.976,A -85,B 0,C 180,E1 -17458.614,E2 -17458.614} C_VEL
LIN {X 0,Y 288.65,Z 472.774,A -85,B 0,C 180,E1 -17459.791,E2 -17459.791} C_VEL
LIN {X 0,Y 286.421,Z 482.494,A -85,B 0,C 180,E1 -17461.407,E2 -17461.407} C_VEL
LIN {X 0,Y 284.231,Z 490.801,A -85,B 0,C 180,E1 -17463.19,E2 -17463.19} C_VEL
LIN {X 0,Y 282.489,Z 496.918,A -85,B 0,C 180,E1 -17464.822,E2 -17464.822} C_VEL
LIN {X 0,Y 280.925,Z 501.911,A -85,B 0,C 180,E1 -17466.465,E2 -17466.465} C_VEL
LIN {X 0,Y 279.795,Z 505.543,A -85,B 0,C 180,E1 -17467.942,E2 -17467.942} C_VEL
LIN {X 0,Y 278.359,Z 509.521,A -85,B 0,C 180,E1 -17470.061,E2 -17470.061} C_VEL
LIN {X 0,Y 277.47,Z 511.757,A -85,B 0,C 180,E1 -17471.692,E2 -17471.692} C_VEL
LIN {X 0,Y 276.796,Z 513.258,A -85,B 0,C 180,E1 -17473.21,E2 -17473.21} C_VEL
LIN {X 0,Y 276.236,Z 514.19,A -85,B 0,C 180,E1 -17474.816,E2 -17474.816} C_VEL
LIN {X 0,Y 275.857,Z 514.417,A -85,B 0,C 180,E1 -17476.276,E2 -17476.276} C_VEL
LIN {X 0,Y 275.533,Z 514.15,A -85,B 0,C 180,E1 -17477.824,E2 -17477.824} C_VEL
LIN {X 0,Y 275.37,Z 513.339,A -85,B 0,C 180,E1 -17479.378,E2 -17479.378} C_VEL
LIN {X 0,Y 275.296,Z 511.966,A -85,B 0,C 180,E1 -17480.942,E2 -17480.942} C_VEL
LIN {X 0,Y 275.369,Z 509.951,A -85,B 0,C 180,E1 -17482.51,E2 -17482.51} C_VEL
LIN {X 0,Y 275.676,Z 505.553,A -85,B 0,C 180,E1 -17484.876,E2 -17484.876} C_VEL
LIN {X 0,Y 276.063,Z 500.181,A -85,B 0,C 180,E1 -17487.002,E2 -17487.002} C_VEL
LIN {X 0,Y 276.496,Z 494.148,A -85,B 0,C 180,E1 -17488.879,E2 -17488.879} C_VEL
LIN {X 0,Y 277.2,Z 486.02,A -85,B 0,C 180,E1 -17490.892,E2 -17490.892} C_VEL
LIN {X 0,Y 277.914,Z 477.71,A -85,B 0,C 180,E1 -17492.506,E2 -17492.506} C_VEL
LIN {X 0,Y 278.667,Z 468.798,A -85,B 0,C 180,E1 -17493.918,E2 -17493.918} C_VEL
LIN {X 0,Y 279.42,Z 459.421,A -85,B 0,C 180,E1 -17495.125,E2 -17495.125} C_VEL
LIN {X 0,Y 280.264,Z 447.49,A -85,B 0,C 180,E1 -17496.331,E2 -17496.331} C_VEL
LIN {X 0,Y 280.842,Z 436.018,A -85,B 0,C 180,E1 -17497.166,E2 -17497.166} C_VEL
LIN {X 0,Y 281.294,Z 426.098,A -85,B 0,C 180,E1 -17497.687,E2 -17497.687} C_VEL
LIN {X 0,Y 283.087,Z 370.175,A -85,B 0,C 180,E1 -17499.683,E2 -17499.683} C_VEL
LIN {X 0,Y 279.628,Z 340.123,A -85,B 0,C 180,E1 -17500.977,E2 -17500.977} C_VEL
LIN {X 0,Y 280.957,Z 328.051,A -85,B 0,C 180,E1 -17504.461,E2 -17504.461} C_VEL
LIN {X 0,Y 280.955,Z 324.432,A -85,B 0,C 180,E1 -17505.542,E2 -17505.542} C_VEL
LIN {X 0,Y 279.067,Z 314.801,A -85,B 0,C 180,E1 -17508.619,E2 -17508.619} C_VEL
LIN {X 0,Y 277.275,Z 305.948,A -85,B 0,C 180,E1 -17511.61,E2 -17511.61} C_VEL
LIN {X 0,Y 277.277,Z 305.943,A -85,B 0,C 180,E1 -17514.341,E2 -17514.341} C_VEL
LIN {X 0,Y 277.239,Z 305.952,A -85,B 0,C 180,E1 -17517.836,E2 -17517.836} C_VEL
LIN {X 0,Y 277.219,Z 305.95,A -85,B 0,C 180,E1 -17521.204,E2 -17521.204} C_VEL
LIN {X 0,Y 277.235,Z 305.952,A -85,B 0,C 180,E1 -17524.471,E2 -17524.471} C_VEL
LIN {X 0,Y 277.252,Z 305.946,A -85,B 0,C 180,E1 -17527.651,E2 -17527.651} C_VEL
LIN {X 0,Y 277.289,Z 305.946,A -85,B 0,C 180,E1 -17530.761,E2 -17530.761} C_VEL
LIN {X 0,Y 277.415,Z 305.926,A -85,B 0,C 180,E1 -17535.323,E2 -17535.323} C_VEL
LIN {X 0,Y 277.46,Z 305.921,A -85,B 0,C 180,E1 -17539.785,E2 -17539.785} C_VEL
LIN {X 0,Y 277.605,Z 305.903,A -85,B 0,C 180,E1 -17542.726,E2 -17542.726} C_VEL
LIN {X 0,Y 277.807,Z 305.877,A -85,B 0,C 180,E1 -17548.548,E2 -17548.548} C_VEL
LIN {X 0,Y 277.806,Z 305.879,A -85,B 0,C 180,E1 -17551.447,E2 -17551.447} C_VEL
LIN {X 0,Y 277.602,Z 305.902,A -85,B 0,C 180,E1 -17557.269,E2 -17557.269} C_VEL
LIN {X 0,Y 277.458,Z 305.925,A -85,B 0,C 180,E1 -17560.209,E2 -17560.209} C_VEL
LIN {X 0,Y 277.408,Z 305.931,A -85,B 0,C 180,E1 -17564.671,E2 -17564.671} C_VEL
LIN {X 0,Y 277.281,Z 305.944,A -85,B 0,C 180,E1 -17569.233,E2 -17569.233} C_VEL
LIN {X 0,Y 277.275,Z 305.943,A -85,B 0,C 180,E1 -17573.92,E2 -17573.92} C_VEL
LIN {X 0,Y 277.26,Z 305.949,A -85,B 0,C 180,E1 -17577.477,E2 -17577.477} C_VEL
LIN {X 0,Y 277.237,Z 305.946,A -85,B 0,C 180,E1 -17580.467,E2 -17580.467} C_VEL
LIN {X 0,Y 277.232,Z 305.952,A -85,B 0,C 180,E1 -17583.89,E2 -17583.89} C_VEL
LIN {X 0,Y 277.241,Z 305.949,A -85,B 0,C 180,E1 -17587.465,E2 -17587.465} C_VEL
LIN {X 0,Y 277.19,Z 305.953,A -85,B 0,C 180,E1 -17591.231,E2 -17591.231} C_VEL
LIN {X 0,Y 277.179,Z 305.955,A -85,B 0,C 180,E1 -17595.221,E2 -17595.221} C_VEL
LIN {X 0,Y 277.193,Z 305.952,A -85,B 0,C 180,E1 -17599.508,E2 -17599.508} C_VEL
LIN {X 0,Y 277.229,Z 305.952,A -85,B 0,C 180,E1 -17602.524,E2 -17602.524} C_VEL
LIN {X 0,Y 277.216,Z 305.95,A -85,B 0,C 180,E1 -17606.099,E2 -17606.099} C_VEL
LIN {X 0,Y 277.231,Z 305.951,A -85,B 0,C 180,E1 -17609.534,E2 -17609.534} C_VEL
LIN {X 0,Y 277.32,Z 305.939,A -85,B 0,C 180,E1 -17612.859,E2 -17612.859} C_VEL
LIN {X 0,Y 277.259,Z 305.945,A -85,B 0,C 180,E1 -17616.072,E2 -17616.072} C_VEL
LIN {X 0,Y 277.243,Z 305.947,A -85,B 0,C 180,E1 -17620.758,E2 -17620.758} C_VEL
LIN {X 0,Y 277.367,Z 305.93,A -85,B 0,C 180,E1 -17625.321,E2 -17625.321} C_VEL
LIN {X 0,Y 277.418,Z 305.927,A -85,B 0,C 180,E1 -17629.785,E2 -17629.785} C_VEL
LIN {X 0,Y 277.591,Z 305.905,A -85,B 0,C 180,E1 -17632.727,E2 -17632.727} C_VEL
LIN {X 0,Y 277.741,Z 305.886,A -85,B 0,C 180,E1 -17638.247,E2 -17638.247} C_VEL
LIN {X 0,Y 277.131,Z 305.967,A -85,B 0,C 180,E1 -17639.458,E2 -17639.458} C_VEL
LIN {X 0,Y 275.491,Z 306.175,A -85,B 0,C 180,E1 -17640.643,E2 -17640.643} C_VEL
LIN {X 0,Y 271.548,Z 306.662,A -85,B 0,C 180,E1 -17643.022,E2 -17643.022} C_VEL
LIN {X 0,Y 270.454,Z 306.793,A -85,B 0,C 180,E1 -17644.267,E2 -17644.267} C_VEL
LIN {X 0,Y 270.379,Z 306.8,A -85,B 0,C 180,E1 -17644.689,E2 -17644.689} C_VEL
LIN {X 0,Y 270.547,Z 306.785,A -85,B 0,C 180,E1 -17647.462,E2 -17647.462} C_VEL
LIN {X 0,Y 270.369,Z 306.802,A -85,B 0,C 180,E1 -17650.483,E2 -17650.483} C_VEL
LIN {X 0,Y 270.341,Z 306.807,A -85,B 0,C 180,E1 -17655.067,E2 -17655.067} C_VEL
LIN {X 0,Y 270.259,Z 306.819,A -85,B 0,C 180,E1 -17659.758,E2 -17659.758} C_VEL
LIN {X 0,Y 270.198,Z 306.828,A -85,B 0,C 180,E1 -17664.592,E2 -17664.592} C_VEL
LIN {X 0,Y 270.207,Z 306.824,A -85,B 0,C 180,E1 -17667.915,E2 -17667.915} C_VEL
LIN {X 0,Y 270.139,Z 306.832,A -85,B 0,C 180,E1 -17671.353,E2 -17671.353} C_VEL
LIN {X 0,Y 270.165,Z 306.834,A -85,B 0,C 180,E1 -17674.91,E2 -17674.91} C_VEL
LIN {X 0,Y 270.168,Z 306.831,A -85,B 0,C 180,E1 -17678.714,E2 -17678.714} C_VEL
LIN {X 0,Y 270.132,Z 306.838,A -85,B 0,C 180,E1 -17683.252,E2 -17683.252} C_VEL
LIN {X 0,Y 270.146,Z 306.836,A -85,B 0,C 180,E1 -17687.446,E2 -17687.446} C_VEL
LIN {X 0,Y 270.185,Z 306.829,A -85,B 0,C 180,E1 -17691.379,E2 -17691.379} C_VEL
LIN {X 0,Y 270.221,Z 306.938,A -85,B 0,C 180,E1 -17695.048,E2 -17695.048} C_VEL
LIN {X 0,Y 273.22,Z 320.363,A -85,B 0,C 180,E1 -17699.046,E2 -17699.046} C_VEL
LIN {X 0,Y 275.87,Z 333.322,A -85,B 0,C 180,E1 -17702.712,E2 -17702.712} C_VEL
LIN {X 0,Y 275.954,Z 335.156,A -85,B 0,C 180,E1 -17703.201,E2 -17703.201} C_VEL
LIN {X 0,Y 274.522,Z 343.899,A -85,B 0,C 180,E1 -17705.423,E2 -17705.423} C_VEL
LIN {X 0,Y 276.482,Z 368.408,A -85,B 0,C 180,E1 -17706.387,E2 -17706.387} C_VEL
LIN {X 0,Y 277.382,Z 379.121,A -85,B 0,C 180,E1 -17706.795,E2 -17706.795} C_VEL
LIN {X 0,Y 275.338,Z 445.858,A -85,B 0,C 180,E1 -17708.97,E2 -17708.97} C_VEL
LIN {X 0,Y 274.838,Z 455.908,A -85,B 0,C 180,E1 -17709.469,E2 -17709.469} C_VEL
LIN {X 0,Y 274.204,Z 464.708,A -85,B 0,C 180,E1 -17710.055,E2 -17710.055} C_VEL
LIN {X 0,Y 273.45,Z 474.303,A -85,B 0,C 180,E1 -17710.876,E2 -17710.876} C_VEL
LIN {X 0,Y 272.599,Z 484.482,A -85,B 0,C 180,E1 -17711.983,E2 -17711.983} C_VEL
LIN {X 0,Y 271.79,Z 492.794,A -85,B 0,C 180,E1 -17713.086,E2 -17713.086} C_VEL
LIN {X 0,Y 270.948,Z 501.023,A -85,B 0,C 180,E1 -17714.393,E2 -17714.393} C_VEL
LIN {X 0,Y 270.294,Z 508.024,A -85,B 0,C 180,E1 -17715.704,E2 -17715.704} C_VEL
LIN {X 0,Y 269.553,Z 516.289,A -85,B 0,C 180,E1 -17717.583,E2 -17717.583} C_VEL
LIN {X 0,Y 269.098,Z 521.887,A -85,B 0,C 180,E1 -17719.09,E2 -17719.09} C_VEL
LIN {X 0,Y 268.753,Z 527.705,A -85,B 0,C 180,E1 -17720.977,E2 -17720.977} C_VEL
LIN {X 0,Y 268.576,Z 533.249,A -85,B 0,C 180,E1 -17723.241,E2 -17723.241} C_VEL
LIN {X 0,Y 268.522,Z 535.993,A -85,B 0,C 180,E1 -17724.583,E2 -17724.583} C_VEL
LIN {X 0,Y 268.436,Z 539.694,A -85,B 0,C 180,E1 -17727.002,E2 -17727.002} C_VEL
LIN {X 0,Y 268.508,Z 541.29,A -85,B 0,C 180,E1 -17728.503,E2 -17728.503} C_VEL
LIN {X 0,Y 268.713,Z 542.452,A -85,B 0,C 180,E1 -17730.003,E2 -17730.003} C_VEL
LIN {X 0,Y 268.355,Z 543.221,A -85,B 0,C 180,E1 -17731.504,E2 -17731.504} C_VEL
LIN {X 0,Y 268.317,Z 543.431,A -85,B 0,C 180,E1 -17733.006,E2 -17733.006} C_VEL
LIN {X 0,Y 268.247,Z 542.72,A -85,B 0,C 180,E1 -17736.018,E2 -17736.018} C_VEL
LIN {X 0,Y 268.662,Z 540.141,A -85,B 0,C 180,E1 -17739.032,E2 -17739.032} C_VEL
LIN {X 0,Y 269.299,Z 537.112,A -85,B 0,C 180,E1 -17741.289,E2 -17741.289} C_VEL
LIN {X 0,Y 270.344,Z 533.025,A -85,B 0,C 180,E1 -17743.533,E2 -17743.533} C_VEL
LIN {X 0,Y 271.928,Z 527.758,A -85,B 0,C 180,E1 -17745.747,E2 -17745.747} C_VEL
LIN {X 0,Y 273.377,Z 522.361,A -85,B 0,C 180,E1 -17747.583,E2 -17747.583} C_VEL
LIN {X 0,Y 274.861,Z 517.339,A -85,B 0,C 180,E1 -17749.019,E2 -17749.019} C_VEL
LIN {X 0,Y 277.004,Z 509.809,A -85,B 0,C 180,E1 -17750.807,E2 -17750.807} C_VEL
LIN {X 0,Y 279.204,Z 501.759,A -85,B 0,C 180,E1 -17752.379,E2 -17752.379} C_VEL
LIN {X 0,Y 281.402,Z 493.209,A -85,B 0,C 180,E1 -17753.749,E2 -17753.749} C_VEL
LIN {X 0,Y 283.491,Z 484.256,A -85,B 0,C 180,E1 -17754.926,E2 -17754.926} C_VEL
LIN {X 0,Y 285.411,Z 474.99,A -85,B 0,C 180,E1 -17755.918,E2 -17755.918} C_VEL
LIN {X 0,Y 287.002,Z 465.571,A -85,B 0,C 180,E1 -17756.741,E2 -17756.741} C_VEL
LIN {X 0,Y 288.652,Z 454.672,A -85,B 0,C 180,E1 -17757.457,E2 -17757.457} C_VEL
LIN {X 0,Y 289.814,Z 445.006,A -85,B 0,C 180,E1 -17757.926,E2 -17757.926} C_VEL
LIN {X 0,Y 291.467,Z 421.916,A -85,B 0,C 180,E1 -17758.734,E2 -17758.734} C_VEL
LIN {X 0,Y 294.192,Z 382.271,A -85,B 0,C 180,E1 -17760.074,E2 -17760.074} C_VEL
LIN {X 0,Y 292.911,Z 369.161,A -85,B 0,C 180,E1 -17760.945,E2 -17760.945} C_VEL
LIN {X 0,Y 291.216,Z 358.256,A -85,B 0,C 180,E1 -17761.839,E2 -17761.839} C_VEL
LIN {X 0,Y 287.345,Z 350.134,A -85,B 0,C 180,E1 -17763.096,E2 -17763.096} C_VEL
LIN {X 0,Y 284.637,Z 345.04,A -85,B 0,C 180,E1 -17764.028,E2 -17764.028} C_VEL
LIN {X 0,Y 283.219,Z 342.109,A -85,B 0,C 180,E1 -17764.577,E2 -17764.577} C_VEL
LIN {X 0,Y 281.347,Z 335.084,A -85,B 0,C 180,E1 -17767.482,E2 -17767.482} C_VEL
LIN {X 0,Y 279.764,Z 329.841,A -85,B 0,C 180,E1 -17769.989,E2 -17769.989} C_VEL
LIN {X 0,Y 277.819,Z 324.506,A -85,B 0,C 180,E1 -17773.079,E2 -17773.079} C_VEL
LIN {X 0,Y 275.945,Z 319.797,A -85,B 0,C 180,E1 -17776.556,E2 -17776.556} C_VEL
LIN {X 0,Y 275.159,Z 317.879,A -85,B 0,C 180,E1 -17778.389,E2 -17778.389} C_VEL
LIN {X 0,Y 274.043,Z 315.07,A -85,B 0,C 180,E1 -17782.013,E2 -17782.013} C_VEL
LIN {X 0,Y 273.66,Z 314.321,A -85,B 0,C 180,E1 -17783.796,E2 -17783.796} C_VEL
LIN {X 0,Y 273.3,Z 313.905,A -85,B 0,C 180,E1 -17788.057,E2 -17788.057} C_VEL
LIN {X 0,Y 273.739,Z 314.497,A -85,B 0,C 180,E1 -17790.804,E2 -17790.804} C_VEL
LIN {X 0,Y 274.206,Z 315.25,A -85,B 0,C 180,E1 -17792.527,E2 -17792.527} C_VEL
LIN {X 0,Y 275.662,Z 318.682,A -85,B 0,C 180,E1 -17796.604,E2 -17796.604} C_VEL
LIN {X 0,Y 277.986,Z 324.136,A -85,B 0,C 180,E1 -17800.813,E2 -17800.813} C_VEL
LIN {X 0,Y 280.077,Z 329.683,A -85,B 0,C 180,E1 -17803.978,E2 -17803.978} C_VEL
LIN {X 0,Y 282.231,Z 336.34,A -85,B 0,C 180,E1 -17807.05,E2 -17807.05} C_VEL
LIN {X 0,Y 283.276,Z 339.802,A -85,B 0,C 180,E1 -17808.388,E2 -17808.388} C_VEL
LIN {X 0,Y 287.373,Z 347.251,A -85,B 0,C 180,E1 -17809.854,E2 -17809.854} C_VEL
LIN {X 0,Y 290.094,Z 352.896,A -85,B 0,C 180,E1 -17810.78,E2 -17810.78} C_VEL
LIN {X 0,Y 292.876,Z 370.979,A -85,B 0,C 180,E1 -17812.383,E2 -17812.383} C_VEL
LIN {X 0,Y 293.807,Z 380.337,A -85,B 0,C 180,E1 -17813.058,E2 -17813.058} C_VEL
LIN {X 0,Y 289.618,Z 430.203,A -85,B 0,C 180,E1 -17815.003,E2 -17815.003} C_VEL
LIN {X 0,Y 288.304,Z 441.808,A -85,B 0,C 180,E1 -17815.668,E2 -17815.668} C_VEL
LIN {X 0,Y 286.509,Z 453.861,A -85,B 0,C 180,E1 -17816.661,E2 -17816.661} C_VEL
LIN {X 0,Y 284.738,Z 463.554,A -85,B 0,C 180,E1 -17817.702,E2 -17817.702} C_VEL
LIN {X 0,Y 282.875,Z 472.4,A -85,B 0,C 180,E1 -17818.88,E2 -17818.88} C_VEL
LIN {X 0,Y 280.76,Z 481.19,A -85,B 0,C 180,E1 -17820.323,E2 -17820.323} C_VEL
LIN {X 0,Y 278.375,Z 490.064,A -85,B 0,C 180,E1 -17822.171,E2 -17822.171} C_VEL
LIN {X 0,Y 276.225,Z 496.945,A -85,B 0,C 180,E1 -17824.013,E2 -17824.013} C_VEL
LIN {X 0,Y 274.385,Z 502.497,A -85,B 0,C 180,E1 -17825.881,E2 -17825.881} C_VEL
LIN {X 0,Y 273.121,Z 506.12,A -85,B 0,C 180,E1 -17827.393,E2 -17827.393} C_VEL
LIN {X 0,Y 272.021,Z 509.09,A -85,B 0,C 180,E1 -17828.919,E2 -17828.919} C_VEL
LIN {X 0,Y 271.067,Z 511.416,A -85,B 0,C 180,E1 -17830.457,E2 -17830.457} C_VEL
LIN {X 0,Y 270.231,Z 513.074,A -85,B 0,C 180,E1 -17832.009,E2 -17832.009} C_VEL
LIN {X 0,Y 269.589,Z 514.18,A -85,B 0,C 180,E1 -17833.57,E2 -17833.57} C_VEL
LIN {X 0,Y 269.042,Z 514.776,A -85,B 0,C 180,E1 -17835.143,E2 -17835.143} C_VEL
LIN {X 0,Y 268.682,Z 514.851,A -85,B 0,C 180,E1 -17836.723,E2 -17836.723} C_VEL
LIN {X 0,Y 268.394,Z 514.31,A -85,B 0,C 180,E1 -17838.315,E2 -17838.315} C_VEL
LIN {X 0,Y 268.243,Z 513.126,A -85,B 0,C 180,E1 -17839.914,E2 -17839.914} C_VEL
LIN {X 0,Y 268.256,Z 510.341,A -85,B 0,C 180,E1 -17842.327,E2 -17842.327} C_VEL
LIN {X 0,Y 268.565,Z 505.94,A -85,B 0,C 180,E1 -17844.753,E2 -17844.753} C_VEL
LIN {X 0,Y 268.836,Z 502.103,A -85,B 0,C 180,E1 -17846.387,E2 -17846.387} C_VEL
LIN {X 0,Y 269.194,Z 497.367,A -85,B 0,C 180,E1 -17848.031,E2 -17848.031} C_VEL
LIN {X 0,Y 269.69,Z 491.584,A -85,B 0,C 180,E1 -17849.679,E2 -17849.679} C_VEL
LIN {X 0,Y 270.26,Z 484.469,A -85,B 0,C 180,E1 -17851.339,E2 -17851.339} C_VEL
LIN {X 0,Y 270.924,Z 476.965,A -85,B 0,C 180,E1 -17852.788,E2 -17852.788} C_VEL
LIN {X 0,Y 271.662,Z 468.593,A -85,B 0,C 180,E1 -17854.124,E2 -17854.124} C_VEL
LIN {X 0,Y 272.353,Z 459.89,A -85,B 0,C 180,E1 -17855.267,E2 -17855.267} C_VEL
LIN {X 0,Y 273.172,Z 448.509,A -85,B 0,C 180,E1 -17856.462,E2 -17856.462} C_VEL
LIN {X 0,Y 273.816,Z 436.691,A -85,B 0,C 180,E1 -17857.358,E2 -17857.358} C_VEL
LIN {X 0,Y 274.264,Z 426.858,A -85,B 0,C 180,E1 -17857.897,E2 -17857.897} C_VEL
LIN {X 0,Y 276.162,Z 371.101,A -85,B 0,C 180,E1 -17859.949,E2 -17859.949} C_VEL
LIN {X 0,Y 272.669,Z 340.204,A -85,B 0,C 180,E1 -17861.317,E2 -17861.317} C_VEL
LIN {X 0,Y 274.135,Z 327.171,A -85,B 0,C 180,E1 -17865.172,E2 -17865.172} C_VEL
LIN {X 0,Y 272.673,Z 318.62,A -85,B 0,C 180,E1 -17867.924,E2 -17867.924} C_VEL
LIN {X 0,Y 270.227,Z 306.824,A -85,B 0,C 180,E1 -17871.972,E2 -17871.972} C_VEL
LIN {X 0,Y 270.216,Z 306.824,A -85,B 0,C 180,E1 -17876.335,E2 -17876.335} C_VEL
LIN {X 0,Y 270.159,Z 306.832,A -85,B 0,C 180,E1 -17880.378,E2 -17880.378} C_VEL
LIN {X 0,Y 270.18,Z 306.829,A -85,B 0,C 180,E1 -17883.755,E2 -17883.755} C_VEL
LIN {X 0,Y 270.185,Z 306.827,A -85,B 0,C 180,E1 -17887.034,E2 -17887.034} C_VEL
LIN {X 0,Y 270.228,Z 306.823,A -85,B 0,C 180,E1 -17890.238,E2 -17890.238} C_VEL
LIN {X 0,Y 270.374,Z 306.806,A -85,B 0,C 180,E1 -17894.932,E2 -17894.932} C_VEL
LIN {X 0,Y 270.412,Z 306.8,A -85,B 0,C 180,E1 -17899.516,E2 -17899.516} C_VEL
LIN {X 0,Y 270.567,Z 306.779,A -85,B 0,C 180,E1 -17902.535,E2 -17902.535} C_VEL
LIN {X 0,Y 270.772,Z 306.753,A -85,B 0,C 180,E1 -17908.51,E2 -17908.51} C_VEL
LIN {X 0,Y 270.771,Z 306.756,A -85,B 0,C 180,E1 -17911.484,E2 -17911.484} C_VEL
LIN {X 0,Y 270.563,Z 306.78,A -85,B 0,C 180,E1 -17917.459,E2 -17917.459} C_VEL
LIN {X 0,Y 270.41,Z 306.801,A -85,B 0,C 180,E1 -17920.478,E2 -17920.478} C_VEL
LIN {X 0,Y 270.367,Z 306.805,A -85,B 0,C 180,E1 -17925.062,E2 -17925.062} C_VEL
LIN {X 0,Y 270.22,Z 306.821,A -85,B 0,C 180,E1 -17929.756,E2 -17929.756} C_VEL
LIN {X 0,Y 270.217,Z 306.823,A -85,B 0,C 180,E1 -17934.585,E2 -17934.585} C_VEL
LIN {X 0,Y 270.189,Z 306.826,A -85,B 0,C 180,E1 -17937.911,E2 -17937.911} C_VEL
LIN {X 0,Y 270.162,Z 306.831,A -85,B 0,C 180,E1 -17941.344,E2 -17941.344} C_VEL
LIN {X 0,Y 270.184,Z 306.827,A -85,B 0,C 180,E1 -17944.9,E2 -17944.9} C_VEL
LIN {X 0,Y 270.181,Z 306.825,A -85,B 0,C 180,E1 -17948.705,E2 -17948.705} C_VEL
LIN {X 0,Y 270.144,Z 306.831,A -85,B 0,C 180,E1 -17953.243,E2 -17953.243} C_VEL
LIN {X 0,Y 270.139,Z 306.831,A -85,B 0,C 180,E1 -17957.434,E2 -17957.434} C_VEL
LIN {X 0,Y 270.182,Z 306.827,A -85,B 0,C 180,E1 -17961.369,E2 -17961.369} C_VEL
LIN {X 0,Y 270.168,Z 306.831,A -85,B 0,C 180,E1 -17965.089,E2 -17965.089} C_VEL
LIN {X 0,Y 270.17,Z 306.833,A -85,B 0,C 180,E1 -17969.126,E2 -17969.126} C_VEL
LIN {X 0,Y 270.232,Z 306.821,A -85,B 0,C 180,E1 -17972.142,E2 -17972.142} C_VEL
LIN {X 0,Y 270.202,Z 306.827,A -85,B 0,C 180,E1 -17975.535,E2 -17975.535} C_VEL
LIN {X 0,Y 270.184,Z 306.828,A -85,B 0,C 180,E1 -17980.235,E2 -17980.235} C_VEL
LIN {X 0,Y 270.327,Z 306.807,A -85,B 0,C 180,E1 -17984.93,E2 -17984.93} C_VEL
LIN {X 0,Y 270.371,Z 306.803,A -85,B 0,C 180,E1 -17989.515,E2 -17989.515} C_VEL
LIN {X 0,Y 270.548,Z 306.784,A -85,B 0,C 180,E1 -17992.536,E2 -17992.536} C_VEL
LIN {X 0,Y 270.746,Z 306.759,A -85,B 0,C 180,E1 -17998.512,E2 -17998.512} C_VEL
LIN {X 0,Y 270.741,Z 306.757,A -85,B 0,C 180,E1 -18001.487,E2 -18001.487} C_VEL
LIN {X 0,Y 270.379,Z 306.8,A -85,B 0,C 180,E1 -18004.689,E2 -18004.689} C_VEL
LIN {X 0,Y 269.748,Z 306.882,A -85,B 0,C 180,E1 -18005.934,E2 -18005.934} C_VEL
LIN {X 0,Y 266.901,Z 307.236,A -85,B 0,C 180,E1 -18007.961,E2 -18007.961} C_VEL
LIN {X 0,Y 264.447,Z 307.544,A -85,B 0,C 180,E1 -18009.61,E2 -18009.61} C_VEL
LIN {X 0,Y 263.373,Z 307.675,A -85,B 0,C 180,E1 -18010.888,E2 -18010.888} C_VEL
LIN {X 0,Y 263.275,Z 307.683,A -85,B 0,C 180,E1 -18011.322,E2 -18011.322} C_VEL
LIN {X 0,Y 263.288,Z 307.688,A -85,B 0,C 180,E1 -18015.481,E2 -18015.481} C_VEL
LIN {X 0,Y 263.223,Z 307.695,A -85,B 0,C 180,E1 -18020.309,E2 -18020.309} C_VEL
LIN {X 0,Y 263.151,Z 307.703,A -85,B 0,C 180,E1 -18025.296,E2 -18025.296} C_VEL
LIN {X 0,Y 263.118,Z 307.708,A -85,B 0,C 180,E1 -18028.736,E2 -18028.736} C_VEL
LIN {X 0,Y 263.093,Z 307.711,A -85,B 0,C 180,E1 -18032.293,E2 -18032.293} C_VEL
LIN {X 0,Y 263.147,Z 307.706,A -85,B 0,C 180,E1 -18036.766,E2 -18036.766} C_VEL
LIN {X 0,Y 263.073,Z 307.714,A -85,B 0,C 180,E1 -18039.877,E2 -18039.877} C_VEL
LIN {X 0,Y 263.075,Z 307.713,A -85,B 0,C 180,E1 -18043.993,E2 -18043.993} C_VEL
LIN {X 0,Y 263.099,Z 307.71,A -85,B 0,C 180,E1 -18048.412,E2 -18048.412} C_VEL
LIN {X 0,Y 263.134,Z 307.709,A -85,B 0,C 180,E1 -18052.107,E2 -18052.107} C_VEL
LIN {X 0,Y 263.22,Z 307.813,A -85,B 0,C 180,E1 -18054.642,E2 -18054.642} C_VEL
LIN {X 0,Y 266.375,Z 322.227,A -85,B 0,C 180,E1 -18059.044,E2 -18059.044} C_VEL
LIN {X 0,Y 268.936,Z 334.817,A -85,B 0,C 180,E1 -18062.685,E2 -18062.685} C_VEL
LIN {X 0,Y 267.623,Z 343.856,A -85,B 0,C 180,E1 -18065.057,E2 -18065.057} C_VEL
LIN {X 0,Y 269.298,Z 366.525,A -85,B 0,C 180,E1 -18065.979,E2 -18065.979} C_VEL
LIN {X 0,Y 270.433,Z 379.757,A -85,B 0,C 180,E1 -18066.5,E2 -18066.5} C_VEL
LIN {X 0,Y 268.372,Z 445.303,A -85,B 0,C 180,E1 -18068.699,E2 -18068.699} C_VEL
LIN {X 0,Y 267.857,Z 455.421,A -85,B 0,C 180,E1 -18069.21,E2 -18069.21} C_VEL
LIN {X 0,Y 267.205,Z 464.252,A -85,B 0,C 180,E1 -18069.811,E2 -18069.811} C_VEL
LIN {X 0,Y 266.498,Z 472.929,A -85,B 0,C 180,E1 -18070.558,E2 -18070.558} C_VEL
LIN {X 0,Y 265.657,Z 483.298,A -85,B 0,C 180,E1 -18071.696,E2 -18071.696} C_VEL
LIN {X 0,Y 264.881,Z 491.422,A -85,B 0,C 180,E1 -18072.777,E2 -18072.777} C_VEL
LIN {X 0,Y 263.953,Z 500.069,A -85,B 0,C 180,E1 -18074.167,E2 -18074.167} C_VEL
LIN {X 0,Y 263.176,Z 508.02,A -85,B 0,C 180,E1 -18075.704,E2 -18075.704} C_VEL
LIN {X 0,Y 262.598,Z 514.773,A -85,B 0,C 180,E1 -18077.249,E2 -18077.249} C_VEL
LIN {X 0,Y 261.998,Z 521.754,A -85,B 0,C 180,E1 -18079.181,E2 -18079.181} C_VEL
LIN {X 0,Y 261.702,Z 526.512,A -85,B 0,C 180,E1 -18080.732,E2 -18080.732} C_VEL
LIN {X 0,Y 261.511,Z 532.23,A -85,B 0,C 180,E1 -18083.058,E2 -18083.058} C_VEL
LIN {X 0,Y 261.48,Z 536.601,A -85,B 0,C 180,E1 -18085.379,E2 -18085.379} C_VEL
LIN {X 0,Y 261.371,Z 538.888,A -85,B 0,C 180,E1 -18086.921,E2 -18086.921} C_VEL
LIN {X 0,Y 261.656,Z 541.845,A -85,B 0,C 180,E1 -18090.003,E2 -18090.003} C_VEL
LIN {X 0,Y 261.275,Z 542.681,A -85,B 0,C 180,E1 -18091.544,E2 -18091.544} C_VEL
LIN {X 0,Y 261.243,Z 542.944,A -85,B 0,C 180,E1 -18093.087,E2 -18093.087} C_VEL
LIN {X 0,Y 261.169,Z 542.654,A -85,B 0,C 180,E1 -18095.347,E2 -18095.347} C_VEL
LIN {X 0,Y 261.31,Z 541.37,A -85,B 0,C 180,E1 -18097.731,E2 -18097.731} C_VEL
LIN {X 0,Y 261.606,Z 540.032,A -85,B 0,C 180,E1 -18099.278,E2 -18099.278} C_VEL
LIN {X 0,Y 262.315,Z 537.144,A -85,B 0,C 180,E1 -18101.594,E2 -18101.594} C_VEL
LIN {X 0,Y 263.441,Z 533.191,A -85,B 0,C 180,E1 -18103.894,E2 -18103.894} C_VEL
LIN {X 0,Y 265.108,Z 528.057,A -85,B 0,C 180,E1 -18106.164,E2 -18106.164} C_VEL
LIN {X 0,Y 266.632,Z 522.869,A -85,B 0,C 180,E1 -18108.043,E2 -18108.043} C_VEL
LIN {X 0,Y 268.645,Z 516.613,A -85,B 0,C 180,E1 -18109.884,E2 -18109.884} C_VEL
LIN {X 0,Y 270.97,Z 509.078,A -85,B 0,C 180,E1 -18111.692,E2 -18111.692} C_VEL
LIN {X 0,Y 273.289,Z 500.955,A -85,B 0,C 180,E1 -18113.291,E2 -18113.291} C_VEL
LIN {X 0,Y 275.647,Z 492.304,A -85,B 0,C 180,E1 -18114.678,E2 -18114.678} C_VEL
LIN {X 0,Y 277.838,Z 483.337,A -85,B 0,C 180,E1 -18115.871,E2 -18115.871} C_VEL
LIN {X 0,Y 279.522,Z 475.809,A -85,B 0,C 180,E1 -18116.707,E2 -18116.707} C_VEL
LIN {X 0,Y 281.396,Z 465.714,A -85,B 0,C 180,E1 -18117.62,E2 -18117.62} C_VEL
LIN {X 0,Y 283.121,Z 455.059,A -85,B 0,C 180,E1 -18118.343,E2 -18118.343} C_VEL
LIN {X 0,Y 284.429,Z 444.702,A -85,B 0,C 180,E1 -18118.855,E2 -18118.855} C_VEL
LIN {X 0,Y 286.152,Z 422.033,A -85,B 0,C 180,E1 -18119.664,E2 -18119.664} C_VEL
LIN {X 0,Y 288.997,Z 383.429,A -85,B 0,C 180,E1 -18121.008,E2 -18121.008} C_VEL
LIN {X 0,Y 287.893,Z 370.943,A -85,B 0,C 180,E1 -18121.876,E2 -18121.876} C_VEL
LIN {X 0,Y 286.474,Z 361.698,A -85,B 0,C 180,E1 -18122.664,E2 -18122.664} C_VEL
LIN {X 0,Y 282.075,Z 352.181,A -85,B 0,C 180,E1 -18124.247,E2 -18124.247} C_VEL
LIN {X 0,Y 278.599,Z 346.024,A -85,B 0,C 180,E1 -18125.516,E2 -18125.516} C_VEL
LIN {X 0,Y 276.433,Z 341.965,A -85,B 0,C 180,E1 -18126.437,E2 -18126.437} C_VEL
LIN {X 0,Y 274.419,Z 334.851,A -85,B 0,C 180,E1 -18129.81,E2 -18129.81} C_VEL
LIN {X 0,Y 272.634,Z 329.655,A -85,B 0,C 180,E1 -18132.85,E2 -18132.85} C_VEL
LIN {X 0,Y 271.219,Z 325.842,A -85,B 0,C 180,E1 -18135.603,E2 -18135.603} C_VEL
LIN {X 0,Y 270.43,Z 323.663,A -85,B 0,C 180,E1 -18137.493,E2 -18137.493} C_VEL
LIN {X 0,Y 269.066,Z 320.38,A -85,B 0,C 180,E1 -18141.589,E2 -18141.589} C_VEL
LIN {X 0,Y 268.549,Z 319.25,A -85,B 0,C 180,E1 -18144.218,E2 -18144.218} C_VEL
LIN {X 0,Y 268.349,Z 319.022,A -85,B 0,C 180,E1 -18148.414,E2 -18148.414} C_VEL
LIN {X 0,Y 269.035,Z 320.017,A -85,B 0,C 180,E1 -18151.953,E2 -18151.953} C_VEL
LIN {X 0,Y 270.129,Z 322.684,A -85,B 0,C 180,E1 -18155.583,E2 -18155.583} C_VEL
LIN {X 0,Y 271.543,Z 326.213,A -85,B 0,C 180,E1 -18158.757,E2 -18158.757} C_VEL
LIN {X 0,Y 272.995,Z 329.671,A -85,B 0,C 180,E1 -18161.23,E2 -18161.23} C_VEL
LIN {X 0,Y 275.038,Z 335.376,A -85,B 0,C 180,E1 -18164.454,E2 -18164.454} C_VEL
LIN {X 0,Y 276.474,Z 339.981,A -85,B 0,C 180,E1 -18166.536,E2 -18166.536} C_VEL
LIN {X 0,Y 280.515,Z 346.891,A -85,B 0,C 180,E1 -18168.141,E2 -18168.141} C_VEL
LIN {X 0,Y 283.407,Z 352.17,A -85,B 0,C 180,E1 -18169.21,E2 -18169.21} C_VEL
LIN {X 0,Y 285.539,Z 357.01,A -85,B 0,C 180,E1 -18170.029,E2 -18170.029} C_VEL
LIN {X 0,Y 287.906,Z 373.64,A -85,B 0,C 180,E1 -18171.523,E2 -18171.523} C_VEL
LIN {X 0,Y 288.647,Z 381.011,A -85,B 0,C 180,E1 -18172.102,E2 -18172.102} C_VEL
LIN {X 0,Y 284.238,Z 430.546,A -85,B 0,C 180,E1 -18174.085,E2 -18174.085} C_VEL
LIN {X 0,Y 282.753,Z 442.934,A -85,B 0,C 180,E1 -18174.808,E2 -18174.808} C_VEL
LIN {X 0,Y 280.73,Z 455.347,A -85,B 0,C 180,E1 -18175.873,E2 -18175.873} C_VEL
LIN {X 0,Y 279.177,Z 463.378,A -85,B 0,C 180,E1 -18176.754,E2 -18176.754} C_VEL
LIN {X 0,Y 277.078,Z 472.624,A -85,B 0,C 180,E1 -18178.002,E2 -18178.002} C_VEL
LIN {X 0,Y 274.945,Z 480.899,A -85,B 0,C 180,E1 -18179.384,E2 -18179.384} C_VEL
LIN {X 0,Y 272.599,Z 489.305,A -85,B 0,C 180,E1 -18181.108,E2 -18181.108} C_VEL
LIN {X 0,Y 270.239,Z 496.493,A -85,B 0,C 180,E1 -18182.982,E2 -18182.982} C_VEL
LIN {X 0,Y 268.087,Z 502.58,A -85,B 0,C 180,E1 -18185.039,E2 -18185.039} C_VEL
LIN {X 0,Y 266.492,Z 506.724,A -85,B 0,C 180,E1 -18186.816,E2 -18186.816} C_VEL
LIN {X 0,Y 264.78,Z 510.807,A -85,B 0,C 180,E1 -18189.165,E2 -18189.165} C_VEL
LIN {X 0,Y 263.822,Z 512.791,A -85,B 0,C 180,E1 -18190.748,E2 -18190.748} C_VEL
LIN {X 0,Y 262.991,Z 514.235,A -85,B 0,C 180,E1 -18192.345,E2 -18192.345} C_VEL
LIN {X 0,Y 262.358,Z 515.102,A -85,B 0,C 180,E1 -18193.952,E2 -18193.952} C_VEL
LIN {X 0,Y 261.861,Z 515.326,A -85,B 0,C 180,E1 -18195.569,E2 -18195.569} C_VEL
LIN {X 0,Y 261.486,Z 515.015,A -85,B 0,C 180,E1 -18197.197,E2 -18197.197} C_VEL
LIN {X 0,Y 261.17,Z 513.55,A -85,B 0,C 180,E1 -18199.644,E2 -18199.644} C_VEL
LIN {X 0,Y 261.14,Z 510.73,A -85,B 0,C 180,E1 -18202.135,E2 -18202.135} C_VEL
LIN {X 0,Y 261.46,Z 506.311,A -85,B 0,C 180,E1 -18204.623,E2 -18204.623} C_VEL
LIN {X 0,Y 261.713,Z 502.448,A -85,B 0,C 180,E1 -18206.302,E2 -18206.302} C_VEL
LIN {X 0,Y 262.135,Z 496.955,A -85,B 0,C 180,E1 -18208.214,E2 -18208.214} C_VEL
LIN {X 0,Y 262.568,Z 491.889,A -85,B 0,C 180,E1 -18209.683,E2 -18209.683} C_VEL
LIN {X 0,Y 263.113,Z 485.324,A -85,B 0,C 180,E1 -18211.271,E2 -18211.271} C_VEL
LIN {X 0,Y 263.845,Z 477.31,A -85,B 0,C 180,E1 -18212.87,E2 -18212.87} C_VEL
LIN {X 0,Y 264.549,Z 469.327,A -85,B 0,C 180,E1 -18214.189,E2 -18214.189} C_VEL
LIN {X 0,Y 265.259,Z 460.835,A -85,B 0,C 180,E1 -18215.35,E2 -18215.35} C_VEL
LIN {X 0,Y 265.984,Z 450.641,A -85,B 0,C 180,E1 -18216.479,E2 -18216.479} C_VEL
LIN {X 0,Y 266.775,Z 437.981,A -85,B 0,C 180,E1 -18217.52,E2 -18217.52} C_VEL
LIN {X 0,Y 267.282,Z 427.096,A -85,B 0,C 180,E1 -18218.142,E2 -18218.142} C_VEL
LIN {X 0,Y 269.166,Z 371.156,A -85,B 0,C 180,E1 -18220.266,E2 -18220.266} C_VEL
LIN {X 0,Y 265.695,Z 340.344,A -85,B 0,C 180,E1 -18221.651,E2 -18221.651} C_VEL
LIN {X 0,Y 267.134,Z 328.381,A -85,B 0,C 180,E1 -18225.264,E2 -18225.264} C_VEL
LIN {X 0,Y 265.752,Z 320.135,A -85,B 0,C 180,E1 -18227.971,E2 -18227.971} C_VEL
LIN {X 0,Y 263.198,Z 307.698,A -85,B 0,C 180,E1 -18232.27,E2 -18232.27} C_VEL
LIN {X 0,Y 263.154,Z 307.706,A -85,B 0,C 180,E1 -18235.886,E2 -18235.886} C_VEL
LIN {X 0,Y 263.112,Z 307.709,A -85,B 0,C 180,E1 -18239.502,E2 -18239.502} C_VEL
LIN {X 0,Y 263.115,Z 307.708,A -85,B 0,C 180,E1 -18242.994,E2 -18242.994} C_VEL
LIN {X 0,Y 263.12,Z 307.712,A -85,B 0,C 180,E1 -18246.38,E2 -18246.38} C_VEL
LIN {X 0,Y 263.213,Z 307.695,A -85,B 0,C 180,E1 -18249.688,E2 -18249.688} C_VEL
LIN {X 0,Y 263.316,Z 307.684,A -85,B 0,C 180,E1 -18254.518,E2 -18254.518} C_VEL
LIN {X 0,Y 263.352,Z 307.682,A -85,B 0,C 180,E1 -18259.231,E2 -18259.231} C_VEL
LIN {X 0,Y 263.531,Z 307.655,A -85,B 0,C 180,E1 -18262.335,E2 -18262.335} C_VEL
LIN {X 0,Y 263.736,Z 307.63,A -85,B 0,C 180,E1 -18268.47,E2 -18268.47} C_VEL
LIN {X 0,Y 263.735,Z 307.632,A -85,B 0,C 180,E1 -18271.524,E2 -18271.524} C_VEL
LIN {X 0,Y 263.527,Z 307.657,A -85,B 0,C 180,E1 -18277.659,E2 -18277.659} C_VEL
LIN {X 0,Y 263.353,Z 307.678,A -85,B 0,C 180,E1 -18280.762,E2 -18280.762} C_VEL
LIN {X 0,Y 263.309,Z 307.683,A -85,B 0,C 180,E1 -18285.476,E2 -18285.476} C_VEL
LIN {X 0,Y 263.205,Z 307.696,A -85,B 0,C 180,E1 -18290.306,E2 -18290.306} C_VEL
LIN {X 0,Y 263.16,Z 307.706,A -85,B 0,C 180,E1 -18295.29,E2 -18295.29} C_VEL
LIN {X 0,Y 263.12,Z 307.707,A -85,B 0,C 180,E1 -18298.73,E2 -18298.73} C_VEL
LIN {X 0,Y 263.115,Z 307.707,A -85,B 0,C 180,E1 -18302.283,E2 -18302.283} C_VEL
LIN {X 0,Y 263.161,Z 307.701,A -85,B 0,C 180,E1 -18306.756,E2 -18306.756} C_VEL
LIN {X 0,Y 263.088,Z 307.713,A -85,B 0,C 180,E1 -18309.867,E2 -18309.867} C_VEL
LIN {X 0,Y 263.083,Z 307.714,A -85,B 0,C 180,E1 -18313.983,E2 -18313.983} C_VEL
LIN {X 0,Y 263.095,Z 307.712,A -85,B 0,C 180,E1 -18318.403,E2 -18318.403} C_VEL
LIN {X 0,Y 263.131,Z 307.706,A -85,B 0,C 180,E1 -18322.097,E2 -18322.097} C_VEL
LIN {X 0,Y 263.124,Z 307.705,A -85,B 0,C 180,E1 -18325.88,E2 -18325.88} C_VEL
LIN {X 0,Y 263.119,Z 307.709,A -85,B 0,C 180,E1 -18329.502,E2 -18329.502} C_VEL
LIN {X 0,Y 263.156,Z 307.704,A -85,B 0,C 180,E1 -18332.998,E2 -18332.998} C_VEL
LIN {X 0,Y 263.115,Z 307.705,A -85,B 0,C 180,E1 -18336.38,E2 -18336.38} C_VEL
LIN {X 0,Y 263.171,Z 307.705,A -85,B 0,C 180,E1 -18339.685,E2 -18339.685} C_VEL
LIN {X 0,Y 263.27,Z 307.687,A -85,B 0,C 180,E1 -18344.516,E2 -18344.516} C_VEL
LIN {X 0,Y 263.31,Z 307.683,A -85,B 0,C 180,E1 -18349.231,E2 -18349.231} C_VEL
LIN {X 0,Y 263.51,Z 307.662,A -85,B 0,C 180,E1 -18352.336,E2 -18352.336} C_VEL
LIN {X 0,Y 263.711,Z 307.635,A -85,B 0,C 180,E1 -18358.472,E2 -18358.472} C_VEL
LIN {X 0,Y 263.706,Z 307.633,A -85,B 0,C 180,E1 -18361.526,E2 -18361.526} C_VEL
LIN {X 0,Y 263.509,Z 307.66,A -85,B 0,C 180,E1 -18367.663,E2 -18367.663} C_VEL
LIN {X 0,Y 263.275,Z 307.683,A -85,B 0,C 180,E1 -18371.322,E2 -18371.322} C_VEL
LIN {X 0,Y 262.579,Z 307.773,A -85,B 0,C 180,E1 -18372.599,E2 -18372.599} C_VEL
LIN {X 0,Y 259.707,Z 308.132,A -85,B 0,C 180,E1 -18374.68,E2 -18374.68} C_VEL
LIN {X 0,Y 257.276,Z 308.437,A -85,B 0,C 180,E1 -18376.372,E2 -18376.372} C_VEL
LIN {X 0,Y 256.221,Z 308.569,A -85,B 0,C 180,E1 -18377.685,E2 -18377.685} C_VEL
LIN {X 0,Y 256.128,Z 308.576,A -85,B 0,C 180,E1 -18378.13,E2 -18378.13} C_VEL
